# B&R Automation Studio project MotionTestBenchMaster (part 33)

#### HmiVariablesBrowse.st
```iecst
ACTION HmiVariablesBrowse:
	CASE VAR_Level OF
		0:
			memset(ADR(HMI_CFG_Display), 0, SIZEOF(HMI_CFG_Display));
			VAR_Level := 5;

		5:
			VAR_VariableName := VAR_InitialVariableName;

			IF VAR_VariableName <> '' THEN
				VAR_Level := 6;
			ELSE
				IF (AID.DataOut.ProjectType = CST_AID_ProjectMachine) THEN
					HMI_CFG_Display[1].Name := 'CFG_Cap_Par';
					HMI_CFG_Display[1].Visibility := TRUE;
				END_IF

				HMI_CFG_Display[2].Name := 'CFG_ITC';
				HMI_CFG_Display[2].Visibility := TRUE;

				HMI_CFG_Display[10].Name := 'CFG_Par';
				HMI_CFG_Display[10].Visibility := TRUE;
			END_IF

			IF HMI_CFG_Selection <> 0 THEN
				VAR_InitialVariableName := HMI_CFG_Display[HMI_CFG_Selection].Name;
			END_IF

		6:
			VAR_Page := 0;
			VAR_LastElementOld := 0;
			VAR_LastElement := 0;
			VAR_Level := 7;

		7:
			memset(ADR(HMI_CFG_Display), 0, SIZEOF(HMI_CFG_Display));

			IF VAR_InitialVariableName = 'CFG_Par' THEN
				VAR_Level := 8;
			ELSE
				VAR_Level := 9;
			END_IF

		8:
			HMI_CFG_Display[1].Visibility := TRUE;
			HMI_CFG_Display[1].Name := 'CFG_Par';

			VAR_Level := 100;

		9:
			VAR_PV_NinfoState := PV_ninfo(ADR(VAR_VariableName), ADR(VAR_DType), ADR(VAR_Len), ADR(VAR_Dim));

			IF VAR_Dim <= 20 THEN
				FOR var_i := 1 TO VAR_Dim DO
					PV_item(ADR(VAR_VariableName), UDINT_TO_UINT(var_i - 1), ADR(VAR_ItemName));
					strcat(ADR(HMI_CFG_Display[var_i].Name), ADR(VAR_VariableName));
					strcat(ADR(HMI_CFG_Display[var_i].Name), ADR('.'));
					strcat(ADR(HMI_CFG_Display[var_i].Name), ADR(VAR_ItemName));
					HMI_CFG_Display[var_i].Visibility := TRUE;
				END_FOR
			ELSE
				FOR var_i := 1 TO 20 DO
					IF var_i = 1 AND VAR_Page <> 0 THEN
						HMI_CFG_Display[1].Name := 'Previous elements';
						HMI_CFG_Display[1].Visibility := TRUE;
					ELSIF var_i = 20 AND VAR_Dim > INT_TO_UINT(VAR_LastElement) THEN
						HMI_CFG_Display[20].Name := 'Next elements';
						HMI_CFG_Display[20].Visibility := TRUE;
					ELSIF (var_i + (VAR_Page * VAR_LastElementOld)) <= VAR_Dim THEN
						PV_item(ADR(VAR_VariableName), UDINT_TO_UINT((var_i + (VAR_Page * VAR_LastElementOld)) - 1), ADR(VAR_ItemName));
						strcat(ADR(HMI_CFG_Display[var_i].Name), ADR(VAR_VariableName));
						strcat(ADR(HMI_CFG_Display[var_i].Name), ADR('.'));
						strcat(ADR(HMI_CFG_Display[var_i].Name), ADR(VAR_ItemName));
						HMI_CFG_Display[var_i].Visibility := TRUE;
						VAR_LastElement := UDINT_TO_INT(var_i) + (VAR_Page * VAR_LastElementOld);
					END_IF
				END_FOR
			END_IF
			VAR_LastElementOld := VAR_LastElement;

			VAR_Level := 10;

		10:
			IF HMI_CFG_Selection <> 0 AND
				(NOT HMI_CFG_Display[HMI_CFG_Selection].PresentB	AND NOT HMI_CFG_Display[HMI_CFG_Selection].PresentI		AND
				NOT HMI_CFG_Display[HMI_CFG_Selection].PresentR		AND NOT HMI_CFG_Display[HMI_CFG_Selection].PresentSt)	THEN
				IF VAR_Dim <= 20 THEN
					VAR_Level := 15;
				ELSIF HMI_CFG_Selection = 1 AND VAR_Page <> 0 THEN
					VAR_Level := 7;
				ELSIF HMI_CFG_Selection = 20 AND VAR_Dim > INT_TO_UINT(VAR_LastElement) THEN
					VAR_Level := 7;
				ELSE
					VAR_Level := 15;
				END_IF
			END_IF

		15:
			VAR_Page := 0;
			VAR_LastElementOld := 0;
			VAR_LastElement := 0;
			VAR_Level := 16;

		16:
			memset(ADR(HMI_CFG_Display), 0, SIZEOF(HMI_CFG_Display));
			VAR_Level := 20;

		20:
			VAR_PV_NinfoState := PV_ninfo(ADR(VAR_VariableName), ADR(VAR_DType), ADR(VAR_Len), ADR(VAR_Dim));

			IF VAR_DType = 0 THEN
				IF VAR_Dim <= 20 THEN
					FOR var_i := 1 TO VAR_Dim DO
						PV_item(ADR(VAR_VariableName), UDINT_TO_UINT(var_i - 1), ADR(VAR_ItemName));
						strcat(ADR(HMI_CFG_Display[var_i].Name), ADR(VAR_VariableName));
						strcat(ADR(HMI_CFG_Display[var_i].Name), ADR('.'));
						strcat(ADR(HMI_CFG_Display[var_i].Name), ADR(VAR_ItemName));
						HMI_CFG_Display[var_i].Visibility := TRUE;
						VAR_PV_NinfoState := PV_ninfo(ADR(HMI_CFG_Display[var_i].Name), ADR(VAR_DType2), ADR(VAR_Len2), ADR(VAR_Dim2));
						IF VAR_DType2 = 1 THEN
							PV_xgetadr(ADR(HMI_CFG_Display[var_i].Name), ADR(VAR_address), ADR(VAR_Len2));
							memcpy(ADR(HMI_CFG_Display[var_i].ValueB), VAR_address, VAR_Len2);
							HMI_CFG_Display[var_i].PresentB := TRUE;
						ELSIF (VAR_DType2 >= 2 AND VAR_DType2 <= 7) OR VAR_DType2 = 12 THEN
							PV_xgetadr(ADR(HMI_CFG_Display[var_i].Name), ADR(VAR_address), ADR(VAR_Len2));
							memcpy(ADR(HMI_CFG_Display[var_i].ValueI), VAR_address, VAR_Len2);
							HMI_CFG_Display[var_i].PresentI := TRUE;
						ELSIF VAR_DType2 = 8 THEN
							PV_xgetadr(ADR(HMI_CFG_Display[var_i].Name), ADR(VAR_address), ADR(VAR_Len2));
							memcpy(ADR(HMI_CFG_Display[var_i].ValueR), VAR_address, VAR_Len2);
							HMI_CFG_Display[var_i].PresentR := TRUE;
						ELSIF VAR_DType2 = 9 THEN
							PV_xgetadr(ADR(HMI_CFG_Display[var_i].Name), ADR(VAR_address), ADR(VAR_Len2));
							strcpy(ADR(HMI_CFG_Display[var_i].ValueSt), VAR_address);
							HMI_CFG_Display[var_i].PresentSt := TRUE;
						END_IF
					END_FOR
				ELSE
					FOR var_i := 1 TO 20 DO
						IF var_i = 1 AND VAR_Page <> 0 THEN
							HMI_CFG_Display[1].Name := 'Previous elements';
							HMI_CFG_Display[1].Visibility := TRUE;
						ELSIF var_i = 20 AND VAR_Dim > INT_TO_UINT(VAR_LastElement) THEN
							HMI_CFG_Display[20].Name := 'Next elements';
							HMI_CFG_Display[20].Visibility := TRUE;
						ELSIF (var_i + (VAR_Page * VAR_LastElementOld)) <= VAR_Dim THEN
							PV_item(ADR(VAR_VariableName), UDINT_TO_UINT((var_i + (VAR_Page * VAR_LastElementOld)) - 1), ADR(VAR_ItemName));
							strcat(ADR(HMI_CFG_Display[var_i].Name), ADR(VAR_VariableName));
							strcat(ADR(HMI_CFG_Display[var_i].Name), ADR('.'));
							strcat(ADR(HMI_CFG_Display[var_i].Name), ADR(VAR_ItemName));
							HMI_CFG_Display[var_i].Visibility := TRUE;
							VAR_PV_NinfoState := PV_ninfo(ADR(HMI_CFG_Display[var_i].Name), ADR(VAR_DType2), ADR(VAR_Len2), ADR(VAR_Dim2));
							IF VAR_DType2 = 1 THEN
								PV_xgetadr(ADR(HMI_CFG_Display[var_i].Name), ADR(VAR_address), ADR(VAR_Len2));
								memcpy(ADR(HMI_CFG_Display[var_i].ValueB), VAR_address, VAR_Len2);
								HMI_CFG_Display[var_i].PresentB := TRUE;
							ELSIF VAR_DType2 >= 2 AND VAR_DType2 <= 7 OR VAR_DType2 = 12 THEN
								PV_xgetadr(ADR(HMI_CFG_Display[var_i].Name), ADR(VAR_address), ADR(VAR_Len2));
								memcpy(ADR(HMI_CFG_Display[var_i].ValueI), VAR_address, VAR_Len2);
								HMI_CFG_Display[var_i].PresentI := TRUE;
							ELSIF VAR_DType2 = 8 THEN
								PV_xgetadr(ADR(HMI_CFG_Display[var_i].Name), ADR(VAR_address), ADR(VAR_Len2));
								memcpy(ADR(HMI_CFG_Display[var_i].ValueR), VAR_address, VAR_Len2);
								HMI_CFG_Display[var_i].PresentR := TRUE;
							ELSIF VAR_DType2 = 9 THEN
								PV_xgetadr(ADR(HMI_CFG_Display[var_i].Name), ADR(VAR_address), ADR(VAR_Len2));
								strcpy(ADR(HMI_CFG_Display[var_i].ValueSt), VAR_address);
								HMI_CFG_Display[var_i].PresentSt := TRUE;
							END_IF
							VAR_LastElement := UDINT_TO_INT(var_i) + (VAR_Page * VAR_LastElementOld);
						END_IF
					END_FOR
				END_IF
			ELSIF VAR_DType = 15 THEN
				FOR var_i := 1 TO VAR_Dim DO
					strcat(ADR(HMI_CFG_Display[var_i].Name), ADR(VAR_VariableName));
					strcat(ADR(HMI_CFG_Display[var_i].Name), ADR('['));
					itoa((var_i - 1), ADR(VAR_array));
					strcat(ADR(HMI_CFG_Display[var_i].Name), ADR(VAR_array));
					strcat(ADR(HMI_CFG_Display[var_i].Name), ADR(']'));
					HMI_CFG_Display[var_i].Visibility := TRUE;
				END_FOR
			END_IF
			VAR_LastElementOld := VAR_LastElement;

			VAR_Level := 30;

		30:
			IF HMI_CFG_Selection <> 0 AND
				(NOT HMI_CFG_Display[HMI_CFG_Selection].PresentB	AND NOT HMI_CFG_Display[HMI_CFG_Selection].PresentI		AND
				NOT HMI_CFG_Display[HMI_CFG_Selection].PresentR		AND NOT HMI_CFG_Display[HMI_CFG_Selection].PresentSt)	THEN
				IF VAR_Dim <= 20 THEN
					VAR_Level := 15;
				ELSIF HMI_CFG_Selection = 1 AND VAR_Page <> 0 THEN
					VAR_Level := 16;
				ELSIF HMI_CFG_Selection = 20 AND VAR_Dim > INT_TO_UINT(VAR_LastElement) THEN
					VAR_Level := 16;
				ELSE
					VAR_Level := 15;
				END_IF
			END_IF

			FOR var_i := 1 TO 20 DO
				IF HMI_CFG_Display[var_i].PresentB THEN
					PV_xgetadr(ADR(HMI_CFG_Display[var_i].Name), ADR(VAR_address), ADR(VAR_Len2));
					memcpy(VAR_address, ADR(HMI_CFG_Display[var_i].ValueB), VAR_Len2);
				ELSIF HMI_CFG_Display[var_i].PresentI THEN
					PV_xgetadr(ADR(HMI_CFG_Display[var_i].Name), ADR(VAR_address), ADR(VAR_Len2));
					memcpy(VAR_address, ADR(HMI_CFG_Display[var_i].ValueI), VAR_Len2);
				ELSIF HMI_CFG_Display[var_i].PresentR THEN
					PV_xgetadr(ADR(HMI_CFG_Display[var_i].Name), ADR(VAR_address), ADR(VAR_Len2));
					memcpy(VAR_address, ADR(HMI_CFG_Display[var_i].ValueR), VAR_Len2);
				ELSIF HMI_CFG_Display[var_i].PresentSt THEN
					PV_xgetadr(ADR(HMI_CFG_Display[var_i].Name), ADR(VAR_address), ADR(VAR_Len2));
					strcpy(VAR_address, ADR(HMI_CFG_Display[var_i].ValueSt));
				ELSE
					EXIT;
				END_IF
			END_FOR
	END_CASE

	IF EDGENEG(HMI_CFG_Reset) THEN
		IF VAR_Level = 10 OR VAR_Level = 100 THEN
			VAR_InitialVariableName := '';
		END_IF
		VAR_Level := 0;
	END_IF

	IF HMI_CFG_Selection <> 0 THEN
		IF (NOT HMI_CFG_Display[HMI_CFG_Selection].PresentB	AND NOT HMI_CFG_Display[HMI_CFG_Selection].PresentI		AND
			NOT HMI_CFG_Display[HMI_CFG_Selection].PresentR		AND NOT HMI_CFG_Display[HMI_CFG_Selection].PresentSt)	THEN
			IF VAR_Dim <= 20 THEN
				VAR_VariableName := HMI_CFG_Display[HMI_CFG_Selection].Name;
			ELSIF HMI_CFG_Selection = 1 AND VAR_Page <> 0 THEN
				VAR_Page := VAR_Page - 1;
			ELSIF HMI_CFG_Selection = 20 AND VAR_Dim > INT_TO_UINT(VAR_LastElement) THEN
				VAR_Page := VAR_Page + 1;
			ELSE
				VAR_VariableName := HMI_CFG_Display[HMI_CFG_Selection].Name;
			END_IF

			HMI_CFG_Selection := 0;
		END_IF
	END_IF
END_ACTION
```

#### CsvManager.st
```iecst
ACTION CsvManager:
	VAR_FmCmd.FolderCreate		:= FALSE;
	VAR_FmCmd.Load				:= FALSE;
	VAR_FmCmd.Save				:= FALSE;
	VAR_FileName				:= '';

	CFG.DataOut.CapSaved		:= FALSE;
	CFG.DataOut.Busy			:= VAR_CsvMngState <> 800;

	CASE VAR_CsvMngState OF
		0:		//Create Folder
			VAR_FmCmd.FolderCreate := NOT VAR_FmAck.CommandError;

			IF VAR_FmAck.CommandDone THEN
				VAR_CsvMngState := 99;
			END_IF

		99:		//Wait idle
			IF StFmState = 0 AND NOT VAR_FmAck.CommandDone THEN
				VAR_CsvMngState	:= 100;
			END_IF

		100:	//Load machine configuration
			VAR_FmCmd.Load	:= TRUE;
			VAR_FileName	:= 'CFG_PAO.csv';

			FB_MpRecipeCsv.Category	:= ADR(VAR_CategoryConfig);

			IF VAR_FmAck.CommandError THEN
				VAR_CsvMngState			:= 110;
			ELSIF VAR_FmAck.CommandDone AND FB_MpRecipeCsv.Info.LastLoadedRecipe = VAR_FileName THEN
				VAR_CfgPaoName			:= VAR_Header.Name;
				CFG.DataOut.CfgDefault	:= (VAR_Header.Name = 'Default Value');
				VAR_CsvMngState			:= 199;
			END_IF

		110:	//Wait errore reset and idle
			IF NOT VAR_FmAck.CommandError AND StFmState = 0 THEN
				VAR_CsvMngState	:= 115;
			END_IF

		115:	//Save default machine configuration
			VAR_FmCmd.Save			:= TRUE;
			VAR_FileName			:= 'CFG_PAO.csv';
			FB_MpRecipeCsv.Header	:= ADR(CST_DefaultHeader);
			FB_MpRecipeCsv.Category	:= ADR(VAR_CategoryConfig);

			IF VAR_FmAck.CommandError THEN
				CFG.DataOut.ErrorSavingCfg	:= TRUE;
				VAR_CsvMngState				:= 116;
			ELSIF VAR_FmAck.CommandDone THEN
				CFG.DataOut.CfgDefault		:= TRUE;
				VAR_CsvMngState				:= 199;
			END_IF

		116:	//Wait error reset
			IF NOT VAR_FmAck.CommandError THEN
				VAR_CsvMngState	:= 199;
			END_IF

		199:	//Wait idle
			IF StFmState = 0 AND NOT VAR_FmAck.CommandDone THEN
				IF (AID.DataOut.ProjectType = CST_AID_ProjectMachine) THEN
					VAR_CsvMngState	:= 200;
				ELSE
					VAR_CsvMngState	:= 300;
				END_IF
			END_IF

		200:	//Load Hmi configuration
			VAR_FmCmd.Load	:= TRUE;
			VAR_FileName	:= 'HMI_PAO.csv';

			FB_MpRecipeCsv.Category	:= ADR(VAR_CategoryHmi);

			IF VAR_FmAck.CommandError THEN
				VAR_CsvMngState			:= 210;
			ELSIF VAR_FmAck.CommandDone AND FB_MpRecipeCsv.Info.LastLoadedRecipe = VAR_FileName THEN
				VAR_HmiPaoName			:= VAR_Header.Name;
				CFG.DataOut.PaoDefault	:= (VAR_Header.Name = 'Default Value');
				VAR_CsvMngState			:= 299;
			END_IF

		210:	//Wait errore reset and idle
			IF NOT VAR_FmAck.CommandError AND StFmState = 0 THEN
				VAR_CsvMngState	:= 215;
			END_IF

		215:	//Save default Hmi configuration
			VAR_FmCmd.Save			:= TRUE;
			VAR_FileName			:= 'HMI_PAO.csv';
			FB_MpRecipeCsv.Header	:= ADR(CST_DefaultHeader);
			FB_MpRecipeCsv.Category	:= ADR(VAR_CategoryHmi);

			IF VAR_FmAck.CommandError THEN
				CFG.DataOut.ErrorSavingPao	:= TRUE;
				VAR_CsvMngState				:= 216;
			ELSIF VAR_FmAck.CommandDone THEN
				CFG.DataOut.PaoDefault		:= TRUE;
				VAR_CsvMngState				:= 299;
			END_IF

		216:	//Wait error reset
			IF NOT VAR_FmAck.CommandError THEN
				VAR_CsvMngState	:= 299;
			END_IF

		299:	//Wait idle
			IF StFmState = 0 AND NOT VAR_FmAck.CommandDone THEN
				VAR_CsvMngState	:= 300;
			END_IF

		300:	//Load Itc configuration
			VAR_FmCmd.Load	:= TRUE;
			VAR_FileName	:= 'CFG_ITC.csv';

			FB_MpRecipeCsv.Category	:= ADR(VAR_CategoryItc);

			IF VAR_FmAck.CommandError THEN
				VAR_CsvMngState			:= 310;
			ELSIF VAR_FmAck.CommandDone AND FB_MpRecipeCsv.Info.LastLoadedRecipe = VAR_FileName THEN
				VAR_CfgItcName			:= VAR_Header.Name;
				CFG.DataOut.ItcDefault	:= (VAR_Header.Name = 'Default Value');
				VAR_CsvMngState			:= 399;
			END_IF

		310:	//Wait errore reset and idle
			IF NOT VAR_FmAck.CommandError AND StFmState = 0 THEN
				VAR_CsvMngState	:= 315;
			END_IF

		315:	//Save default Itc configuration
			VAR_FmCmd.Save			:= TRUE;
			VAR_FileName			:= 'CFG_ITC.csv';
			FB_MpRecipeCsv.Header	:= ADR(CST_DefaultHeader);
			FB_MpRecipeCsv.Category	:= ADR(VAR_CategoryItc);

			IF VAR_FmAck.CommandError THEN
				CFG.DataOut.ErrorSavingItc	:= TRUE;
				VAR_CsvMngState				:= 316;
			ELSIF VAR_FmAck.CommandDone THEN
				CFG.DataOut.ItcDefault		:= TRUE;
				VAR_CsvMngState				:= 399;
			END_IF

		316:	//Wait error reset
			IF NOT VAR_FmAck.CommandError THEN
				VAR_CsvMngState	:= 399;
			END_IF

		399:	//Wait idle
			IF StFmState = 0 AND NOT VAR_FmAck.CommandDone THEN
				IF (AID.DataOut.ProjectType = CST_AID_ProjectMachine) THEN
					IF CFG_Par.Machine.Type.SRMA THEN
						VAR_CsvMngState	:= 500;
					ELSIF CFG_Par.Machine.Type.SRMB OR CFG_Par.Machine.Type.SRMC OR CFG_Par.Machine.Type.SRMH OR CFG_Par.Machine.Type.SRMO THEN
						VAR_CsvMngState	:= 400;
					ELSIF CFG_Par.Machine.Type.SRME THEN
						VAR_CsvMngState	:= 500;
					END_IF
				ELSE
					VAR_CsvMngState	:= 700;
				END_IF
			END_IF

		400:	//Load Cap configuration
			VAR_FmCmd.Load	:= TRUE;
			VAR_FileName	:= 'CFG_CAP.csv';

			FB_MpRecipeCsv.Category	:= ADR(VAR_CategoryCfgCap);

			IF VAR_FmAck.CommandError THEN
				VAR_CsvMngState				:= 410;
			ELSIF VAR_FmAck.CommandDone AND FB_MpRecipeCsv.Info.LastLoadedRecipe = VAR_FileName THEN
				VAR_CfgCapName				:= VAR_Header.Name;
				CFG.DataOut.CfgCapDefault	:= (VAR_Header.Name = 'Default Value');
				VAR_CsvMngState				:= 499;
			END_IF

		410:	//Wait errore reset and idle
			IF NOT VAR_FmAck.CommandError AND StFmState = 0 THEN
				VAR_CsvMngState	:= 415;
			END_IF

		415:	//Save default Cap configuration
			VAR_FmCmd.Save			:= TRUE;
			VAR_FileName			:= 'CFG_CAP.csv';
			FB_MpRecipeCsv.Header	:= ADR(CST_DefaultHeader);
			FB_MpRecipeCsv.Category	:= ADR(VAR_CategoryCfgCap);

			IF VAR_FmAck.CommandError THEN
				CFG.DataOut.ErrorSavingCfgCap	:= TRUE;
				VAR_CsvMngState					:= 416;
			ELSIF VAR_FmAck.CommandDone THEN
				CFG.DataOut.CfgCapDefault		:= TRUE;
				VAR_CsvMngState					:= 499;
			END_IF

		416:	//Wait error reset
			IF NOT VAR_FmAck.CommandError THEN
				VAR_CsvMngState	:= 499;
			END_IF

		499:	//Wait idle
			IF StFmState = 0 AND NOT VAR_FmAck.CommandDone THEN
				VAR_CsvMngState	:= 500;
			END_IF

		500:	//Load Motion configuration
			VAR_FmCmd.Load	:= TRUE;
			VAR_FileName	:= 'CFG_MC.csv';

			FB_MpRecipeCsv.Category	:= ADR(VAR_CategoryMotion);

			IF VAR_FmAck.CommandError THEN
				VAR_CsvMngState			:= 510;
			ELSIF VAR_FmAck.CommandDone AND FB_MpRecipeCsv.Info.LastLoadedRecipe = VAR_FileName THEN
				VAR_CfgMotionName			:= VAR_Header.Name;
				CFG.DataOut.MotionDefault	:= (VAR_Header.Name = 'Default Value');
				VAR_CsvMngState				:= 599;
			END_IF

		510:	//Wait errore reset and idle
			IF NOT VAR_FmAck.CommandError AND StFmState = 0 THEN
				VAR_CsvMngState	:= 515;
			END_IF

		515:	//Save default Motion configuration
			VAR_FmCmd.Save			:= TRUE;
			VAR_FileName			:= 'CFG_MC.csv';
			FB_MpRecipeCsv.Header	:= ADR(CST_DefaultHeader);
			FB_MpRecipeCsv.Category	:= ADR(VAR_CategoryMotion);

			IF VAR_FmAck.CommandError THEN
				CFG.DataOut.ErrorSavingMotion	:= TRUE;
				VAR_CsvMngState					:= 516;
			ELSIF VAR_FmAck.CommandDone THEN
				CFG.DataOut.MotionDefault	:= TRUE;
				VAR_CsvMngState				:= 599;
			END_IF

		516:	//Wait error reset
			IF NOT VAR_FmAck.CommandError THEN
				VAR_CsvMngState	:= 599;
			END_IF

		599:	//Wait idle
			IF StFmState = 0 AND NOT VAR_FmAck.CommandDone THEN
				IF CFG_Par.Machine.Type.SRMA THEN
					VAR_CsvMngState	:= 600;
				ELSIF CFG_Par.Machine.Type.SRMB OR CFG_Par.Machine.Type.SRMC OR CFG_Par.Machine.Type.SRMH OR CFG_Par.Machine.Type.SRMO THEN
					VAR_CsvMngState	:= 600;
				ELSIF CFG_Par.Machine.Type.SRME THEN
					VAR_CsvMngState	:= 700;
				END_IF
			END_IF

		600:	//Load Ops configuration
			VAR_FmCmd.Load	:= TRUE;
			VAR_FileName	:= 'CFG_OPS.csv';

			FB_MpRecipeCsv.Category	:= ADR(VAR_CategoryCfgDoor);

			IF VAR_FmAck.CommandError THEN
				VAR_CsvMngState			:= 610;
			ELSIF VAR_FmAck.CommandDone AND FB_MpRecipeCsv.Info.LastLoadedRecipe = VAR_FileName THEN
				VAR_CfgDoorName			:= VAR_Header.Name;
				CFG.DataOut.OPSDefault	:= (VAR_Header.Name = 'Default Value');
				VAR_CsvMngState				:= 699;
			END_IF

		610:	//Wait errore reset and idle
			IF NOT VAR_FmAck.CommandError AND StFmState = 0 THEN
				VAR_CsvMngState	:= 615;
			END_IF

		615:	//Save default OPS configuration
			VAR_FmCmd.Save			:= TRUE;
			VAR_FileName			:= 'CFG_OPS.csv';
			FB_MpRecipeCsv.Header	:= ADR(CST_DefaultHeader);
			FB_MpRecipeCsv.Category	:= ADR(VAR_CategoryCfgDoor);

			IF VAR_FmAck.CommandError THEN
				CFG.DataOut.ErrorSavingOPS	:= TRUE;
				VAR_CsvMngState					:= 616;
			ELSIF VAR_FmAck.CommandDone THEN
				CFG.DataOut.OPSDefault	:= TRUE;
				VAR_CsvMngState				:= 699;
			END_IF

		616:	//Wait error reset
			IF NOT VAR_FmAck.CommandError THEN
				VAR_CsvMngState	:= 699;
			END_IF

		699:	//Wait idle
			IF StFmState = 0 AND NOT VAR_FmAck.CommandDone THEN
				VAR_CsvMngState	:= 700;
			END_IF

		700:	//Check for error
			IF CFG.DataOut.ErrorSavingCfg OR CFG.DataOut.ErrorSavingItc OR ((CFG.DataOut.ErrorSavingPao OR CFG.DataOut.ErrorSavingCfgCap OR CFG.DataOut.ErrorSavingMotion OR CFG.DataOut.OPSDefault) AND AID.DataOut.ProjectType = CST_AID_ProjectMachine) THEN
				VAR_CsvMngState		:= 9998;
			ELSIF CFG.DataOut.CfgDefault OR CFG.DataOut.ItcDefault OR ((CFG.DataOut.PaoDefault OR CFG.DataOut.CfgCapDefault OR CFG.DataOut.MotionDefault OR CFG.DataOut.OPSDefault) AND AID.DataOut.ProjectType = CST_AID_ProjectMachine) THEN
				VAR_CsvMngState		:= 9999;
			ELSE
				IF (VAR_CfgPaoName = VAR_CfgItcName) AND (((VAR_CfgPaoName = VAR_HmiPaoName) AND (VAR_CfgPaoName = VAR_CfgMotionName) AND
					((VAR_CfgPaoName = VAR_CfgDoorName) OR CFG_Par.Machine.Type.SRME)) OR AID.DataOut.ProjectType = CST_AID_ProjectSkid) THEN
					HMI_MachineId	:= VAR_CfgPaoName;
				ELSE
					HMI_MachineId	:= 'Error Name';
				END_IF
				VAR_CsvMngState		:= 800;
			END_IF

		800:	//Initial Configuration done - Waiting for request
			CFG.DataOut.ConfigLoaded := TRUE;

			IF HMI_PB[PB_CFG_LoadPao].ON THEN
				VAR_CsvMngState		:= 1000;
			ELSIF HMI_PB[PB_CFG_SavePao].ON THEN
				VAR_CsvMngState		:= 1050;
			ELSIF HMI_PB[PB_CFG_LoadCfg].ON THEN
				IF VAR_InitialVariableName = 'CFG_ITC' THEN
					VAR_CsvMngState	:= 1100;
				ELSIF VAR_InitialVariableName = 'CFG_Cap_Par' THEN
					VAR_CsvMngState	:= 1200;
				ELSIF VAR_InitialVariableName = 'CFG_Par' THEN
					VAR_CsvMngState	:= 1300;
				END_IF
			ELSIF HMI_PB[PB_CFG_SaveCfg].ON THEN
				IF VAR_InitialVariableName = 'CFG_ITC' THEN
					VAR_CsvMngState	:= 1150;
				ELSIF VAR_InitialVariableName = 'CFG_Cap_Par' THEN
					VAR_CsvMngState	:= 1250;
				ELSIF VAR_InitialVariableName = 'CFG_Par' THEN
					VAR_CsvMngState	:= 1350;
				END_IF
			ELSIF CAP.DataOut.ConfigSaveReq THEN
				VAR_CsvMngState	:= 1250;
			ELSIF OPS.DataOut.ConfigSaveReq THEN
				VAR_CsvMngState	:= 1450;
			END_IF

		1000:	//Manual - Load Hmi configuration
			VAR_FmCmd.Load	:= TRUE;
			VAR_FileName	:= 'HMI_PAO.csv';

			FB_MpRecipeCsv.Category	:= ADR(VAR_CategoryHmi);

			IF VAR_FmAck.CommandError OR VAR_FmAck.CommandDone THEN
				VAR_CsvMngState := 1010;
			END_IF

		1010:	//Wait errore reset and idle
			IF NOT VAR_FmAck.CommandError AND StFmState = 0 AND NOT HMI_PB[PB_CFG_LoadPao].ON THEN
				VAR_CsvMngState	:= 800;
			END_IF

		1050:	//Manual - Save Hmi configuration
			VAR_FmCmd.Save			:= TRUE;
			VAR_FileName			:= 'HMI_PAO.csv';
			VAR_Header.Name			:= HMI_MachineId;
			FB_MpRecipeCsv.Category	:= ADR(VAR_CategoryHmi);

			IF VAR_FmAck.CommandError OR VAR_FmAck.CommandDone THEN
				VAR_CsvMngState	:= 1060;
			END_IF

		1060:	//Wait errore reset and idle
			IF NOT VAR_FmAck.CommandError AND StFmState = 0 AND NOT HMI_PB[PB_CFG_SavePao].ON THEN
				VAR_CsvMngState	:= 800;
			END_IF

		1100:	//Manual - Load ITC configuration
			VAR_FmCmd.Load	:= TRUE;
			VAR_FileName	:= 'CFG_ITC.csv';

			FB_MpRecipeCsv.Category	:= ADR(VAR_CategoryItc);

			IF VAR_FmAck.CommandError OR VAR_FmAck.CommandDone THEN
				VAR_CsvMngState := 1110;
			END_IF

		1110:	//Wait errore reset and idle
			IF NOT VAR_FmAck.CommandError AND StFmState = 0 AND NOT HMI_PB[PB_CFG_LoadCfg].ON THEN
				VAR_CsvMngState	:= 800;
			END_IF

		1150:	//Manual - Save ITC configuration
			VAR_FmCmd.Save			:= TRUE;
			VAR_FileName			:= 'CFG_ITC.csv';
			VAR_Header.Name			:= HMI_MachineId;
			FB_MpRecipeCsv.Category	:= ADR(VAR_CategoryItc);

			IF VAR_FmAck.CommandError OR VAR_FmAck.CommandDone THEN
				VAR_CsvMngState	:= 1160;
			END_IF

		1160:	//Wait errore reset and idle
			IF NOT VAR_FmAck.CommandError AND StFmState = 0 AND NOT HMI_PB[PB_CFG_SaveCfg].ON THEN
				VAR_CsvMngState	:= 800;
			END_IF

		1200:	//Manual - Load Hmi configuration
			VAR_FmCmd.Load	:= TRUE;
			VAR_FileName	:= 'CFG_CAP.csv';

			FB_MpRecipeCsv.Category	:= ADR(VAR_CategoryCfgCap);

			IF VAR_FmAck.CommandError OR VAR_FmAck.CommandDone THEN
				VAR_CsvMngState := 1210;
			END_IF

		1210:	//Wait errore reset and idle
			IF NOT VAR_FmAck.CommandError AND StFmState = 0 AND NOT HMI_PB[PB_CFG_LoadCfg].ON THEN
				VAR_CsvMngState	:= 800;
			END_IF

		1250:	//Manual - Save Hmi configuration
			VAR_FmCmd.Save			:= TRUE;
			VAR_FileName			:= 'CFG_CAP.csv';
			VAR_Header.Name			:= HMI_MachineId;
			FB_MpRecipeCsv.Category	:= ADR(VAR_CategoryCfgCap);

			IF VAR_FmAck.CommandError OR VAR_FmAck.CommandDone THEN
				VAR_CsvMngState	:= 1260;
			END_IF

		1260:	//Wait errore reset and idle
			CFG.DataOut.CapSaved	:= TRUE;

			IF NOT VAR_FmAck.CommandError AND StFmState = 0 AND NOT HMI_PB[PB_CFG_SaveCfg].ON AND NOT CAP.DataOut.ConfigSaveReq THEN
				VAR_CsvMngState	:= 800;
			END_IF

		1300:	//Manual - Load Hmi configuration
			VAR_FmCmd.Load	:= TRUE;
			VAR_FileName	:= 'CFG_PAO.csv';

			FB_MpRecipeCsv.Category	:= ADR(VAR_CategoryConfig);

			IF VAR_FmAck.CommandError OR VAR_FmAck.CommandDone THEN
				VAR_CsvMngState := 1310;
			END_IF

		1310:	//Wait errore reset and idle
			IF NOT VAR_FmAck.CommandError AND StFmState = 0 AND NOT HMI_PB[PB_CFG_LoadCfg].ON THEN
				VAR_CsvMngState	:= 800;
			END_IF

		1350:	//Manual - Save Hmi configuration
			VAR_FmCmd.Save			:= TRUE;
			VAR_FileName			:= 'CFG_PAO.csv';
			VAR_Header.Name			:= HMI_MachineId;
			FB_MpRecipeCsv.Category	:= ADR(VAR_CategoryConfig);

			IF VAR_FmAck.CommandError OR VAR_FmAck.CommandDone THEN
				VAR_CsvMngState	:= 1360;
			END_IF

		1360:	//Wait errore reset and idle
			IF NOT VAR_FmAck.CommandError AND StFmState = 0 AND NOT HMI_PB[PB_CFG_SaveCfg].ON THEN
				VAR_CsvMngState	:= 800;
			END_IF

		1450:	//Manual - Save Hmi configuration
			VAR_FmCmd.Save			:= TRUE;
			VAR_FileName			:= 'CFG_OPS.csv';
			VAR_Header.Name			:= HMI_MachineId;
			FB_MpRecipeCsv.Category	:= ADR(VAR_CategoryCfgDoor);

			IF VAR_FmAck.CommandError OR VAR_FmAck.CommandDone THEN
				VAR_CsvMngState	:= 1460;
			END_IF

		1460:	//Wait errore reset and idle
			CFG.DataOut.OpsSaved	:= TRUE;

			IF NOT VAR_FmAck.CommandError AND StFmState = 0 AND NOT CAP.DataOut.ConfigSaveReq THEN
				VAR_CsvMngState	:= 800;
			END_IF

		9998:	// Error saving file

		9999:	// Default configuration loaded
	END_CASE
END_ACTION
```

#### FileManager.st
```iecst
ACTION FileManager:
	CASE StFmState OF
		0:		//Wait command
			FB_MpRecipeCsv.LoadType		:= mpRECIPE_CSV_LOAD_ALL;
			FB_MpRecipeCsv.Load			:= FALSE;
			FB_MpRecipeCsv.Save			:= FALSE;
			FB_MpRecipeCsv.ErrorReset	:= FALSE;

			VAR_FmAck.CommandBusy	:= FALSE;
			VAR_FmAck.CommandDone	:= FALSE;
			VAR_FmAck.CommandError	:= FALSE;

			IF FB_MpRecipeCsv.Error THEN
				StFmState	:= 999;
			ELSIF VAR_FmCmd.FolderCreate THEN
				StFmState	:= 100;
			ELSIF VAR_FmCmd.Load THEN
				StFmState	:= 200;
			ELSIF VAR_FmCmd.Save THEN
				StFmState	:= 250;
			END_IF

		100:	//Create Folder
			VAR_FmAck.CommandBusy	:= NOT(VAR_FmAck.CommandDone OR VAR_FmAck.CommandError);

			IF NOT VAR_FmCmd.FolderCreate THEN
				StFmState	:= 0;
			ELSIF VAR_FmAck.CommandBusy THEN
				FB_DirCreate();

				IF FB_DirCreate.status = ERR_OK OR FB_DirCreate.status = fiERR_DIR_ALREADY_EXIST THEN
					VAR_FmAck.CommandDone	:= TRUE;
				ELSIF FB_DirCreate.status <> ERR_FUB_BUSY AND FB_DirCreate.status <> ERR_FUB_ENABLE_FALSE THEN
					VAR_FmAck.CommandError	:= TRUE;
					VAR_FmAck.ErrorCode		:= FB_DirCreate.status;
					VAR_FmAck.ErroreState	:= ERR_FOLDER_CREATE;
				END_IF
			END_IF

		200:	//Load
			VAR_FmAck.CommandBusy	:= NOT(VAR_FmAck.CommandDone OR VAR_FmAck.CommandError);
			FB_MpRecipeCsv.Load		:= TRUE;

			IF EDGEPOS(FB_MpRecipeCsv.Error) THEN
				VAR_FmAck.CommandError	:= TRUE;
				VAR_FmAck.ErrorCode		:= FB_MpRecipeCsv.Info.Diag.StatusID.Code;
				VAR_FmAck.ErroreState	:= ERR_LOAD;
			ELSIF EDGEPOS(FB_MpRecipeCsv.CommandDone) AND NOT FB_MpRecipeCsv.Error THEN
				VAR_FmAck.CommandDone	:= TRUE;
			ELSIF NOT VAR_FmCmd.Load AND (NOT FB_MpRecipeCsv.CommandBusy OR FB_MpRecipeCsv.Error) THEN
				StFmState	:= 0;
			END_IF

		250:	//Save configuration
			VAR_FmAck.CommandBusy	:= NOT(VAR_FmAck.CommandDone OR VAR_FmAck.CommandError);
			FB_MpRecipeCsv.Save		:= TRUE;

				IF EDGEPOS(FB_MpRecipeCsv.Error) THEN
					VAR_FmAck.CommandError	:= TRUE;
					VAR_FmAck.ErrorCode		:= FB_MpRecipeCsv.Info.Diag.StatusID.Code;
					VAR_FmAck.ErroreState	:= ERR_SAVE;
				ELSIF EDGEPOS(FB_MpRecipeCsv.CommandDone) AND NOT FB_MpRecipeCsv.Error THEN
					VAR_FmAck.CommandDone	:= TRUE;
				ELSIF NOT VAR_FmCmd.Save AND (NOT FB_MpRecipeCsv.CommandBusy OR FB_MpRecipeCsv.Error) THEN
					StFmState	:= 0;
				END_IF

		999:	//Error Reset
			FB_MpRecipeCsv.ErrorReset := TRUE;

			IF NOT FB_MpRecipeCsv.Error THEN
				StFmState	:= 0;
			END_IF

	END_CASE
END_ACTION
```

### Package Logical/30_MC - Motion Main Folder

### GlobalVariables.var
```iecst
(*General axis task global interface*)
VAR
	VAR_Machine : ST_Machine;
END_VAR
(*Simulation Variables*)
VAR
	VAR_SimulationOn : BOOL;
END_VAR
(*Machine Master Fast*)
VAR
	fbMachineMasterFast : FB_MasterAxis;
END_VAR
(*Master Module Axis Declaration*)
VAR
	VAR_AxPowerSupply01 : ACP10AXIS_typ;
	VAR_AxPowerSupply02 : ACP10AXIS_typ;
	VAR_AxMachineMaster : ACP10AXIS_typ;
END_VAR
(*Filler Module Axis Declaration*)
VAR
	VAR_AxEncEmul : ACP10AXIS_typ;
	VAR_AxFillerModuleMaster : ACP10AXIS_typ;
	VAR_AxFillerIn10 : ACP10AXIS_typ;
	VAR_AxFillerIn09 : ACP10AXIS_typ;
	VAR_AxFillerIn08 : ACP10AXIS_typ;
	VAR_AxFillerIn07 : ACP10AXIS_typ;
	VAR_AxFillerIn06 : ACP10AXIS_typ;
	VAR_AxFillerIn05 : ACP10AXIS_typ;
	VAR_AxFillerIn04 : ACP10AXIS_typ;
	VAR_AxFillerIn03 : ACP10AXIS_typ;
	VAR_AxFillerIn02 : ACP10AXIS_typ;
	VAR_AxFillerIn01 : ACP10AXIS_typ;
	VAR_AxFillerMain : ACP10AXIS_typ;
	VAR_AxFillerOut01 : ACP10AXIS_typ;
	VAR_AxFillerOut02 : ACP10AXIS_typ;
	VAR_AxFillerOut03 : ACP10AXIS_typ;
	VAR_AxFillerOut04 : ACP10AXIS_typ;
	VAR_AxFillerOut05 : ACP10AXIS_typ;
	VAR_AxFillerOut06 : ACP10AXIS_typ;
END_VAR
(*Inlet Module Axis Declaration*)
VAR
	VAR_AxInletModuleMaster : ACP10AXIS_typ;
	VAR_AxInletIn04 : ACP10AXIS_typ;
	VAR_AxInletIn03 : ACP10AXIS_typ;
	VAR_AxInletIn02 : ACP10AXIS_typ;
	VAR_AxInletIn01 : ACP10AXIS_typ;
	VAR_AxInletMain : ACP10AXIS_typ;
	VAR_AxInletOut01 : ACP10AXIS_typ;
	VAR_AxInletOut02 : ACP10AXIS_typ;
	VAR_AxInletOut03 : ACP10AXIS_typ;
	VAR_AxInletOut04 : ACP10AXIS_typ;
END_VAR
(*Outlet Module Axis Declaration*)
VAR
	VAR_AxOutletModuleMaster : ACP10AXIS_typ;
	VAR_AxOutletIn04 : ACP10AXIS_typ;
	VAR_AxOutletIn03 : ACP10AXIS_typ;
	VAR_AxOutletIn02 : ACP10AXIS_typ;
	VAR_AxOutletIn01 : ACP10AXIS_typ;
	VAR_AxOutletMain : ACP10AXIS_typ;
	VAR_AxOutletOut01 : ACP10AXIS_typ;
	VAR_AxOutletOut02 : ACP10AXIS_typ;
	VAR_AxOutletOut03 : ACP10AXIS_typ;
	VAR_AxOutletOut04 : ACP10AXIS_typ;
END_VAR
(*Modules mapp link*)
VAR
	VAR_SpareLink : MpComIdentType; (*Mapp link to spare axes*)
	VAR_MachineLink : MpComIdentType; (*Mapp link for machine*)
	VAR_MasterModuleLink : MpComIdentType; (*Mapp link for master module*)
	VAR_FillerModuleLink : MpComIdentType; (*Mapp link for filler module*)
	VAR_InletModuleLink : MpComIdentType; (*Mapp link for outlet module*)
	VAR_OutletModuleLink : MpComIdentType; (*Mapp link for outlet module*)
	VAR_MpComLinkToParentSpare : UDINT;
END_VAR
(*DECELERATION*)
VAR
	VAR_EmergencyDec : REAL;
	VAR_ShutDownDec : REAL;
END_VAR
(*CAM*)
VAR
	VAR_xMachineInitDone : BOOL;
	VAR_xInletInitDone : BOOL;
	VAR_xFillerInitDone : BOOL;
	VAR_xOutletInitDone : BOOL;
	VAR_CamInitialized : BOOL; (*//v4.A.A.1.6.7*)
END_VAR
(*INTERCHANGE MOTION*)
VAR
	ITC_Motion : ST_LabellerMotionInterface;
END_VAR
```

### CamConfigurator.var
```iecst
(*Cam Configurator*)
(*Clock A-B*)
VAR CONSTANT
	CST_SubModuleMachineCk : USINT := CST_MasterSubModule; (*0 - Master; 1 - Filler; 2 - Outlet*)
	CST_AxisMachineCk : USINT := CST_ModuleMasterAxis;
	CST_OnPositionCkA : REAL := 0.0;
	CST_OffPositionCkA : REAL := 180.0;
	CST_OnPositionCkB : REAL := 270.0;
	CST_OffPositionCkB : REAL := 90.0;
	CST_OnPositionCkA_Fma : REAL := 10.0;
	CST_OffPositionCkA_Fma : REAL := 190.0;
	CST_OnPositionCkB_Fma : REAL := 100.0;
	CST_OffPositionCkB_Fma : REAL := 280.0;
	CST_AdvTimeCkA : REAL := 0.0;
END_VAR
(*Clock 02*)
VAR CONSTANT
	CST_SubModuleCk02 : USINT := CST_MasterSubModule; (*0 - Master; 1 - Filler; 2 - Outlet*)
	CST_AxisCk02 : USINT := CST_ModuleMasterAxis;
	CST_OnPositionCk02 : REAL := 10.0;
	CST_OffPositionCk02 : REAL := 15.0;
	CST_AdvTimeCk02 : REAL := 0.0;
END_VAR
(*Clock 03*)
VAR CONSTANT
	CST_SubModuleCk03 : USINT := CST_MasterSubModule; (*0 - Master; 1 - Filler; 2 - Outlet*)
	CST_AxisCk03 : USINT := CST_ModuleMasterAxis;
	CST_OnPositionCk03 : REAL := 10.0;
	CST_OffPositionCk03 : REAL := 20.0;
	CST_AdvTimeCk03 : REAL := 0.0;
END_VAR
(*Clock 04*)
VAR CONSTANT
	CST_SubModuleCk04 : USINT := CST_MasterSubModule; (*0 - Master; 1 - Filler; 2 - Outlet*)
	CST_AxisCk04 : USINT := CST_ModuleMasterAxis;
	CST_OnPositionCk04 : REAL := 20.0;
	CST_OffPositionCk04 : REAL := 30.0;
	CST_AdvTimeCk04 : USINT := 0;
END_VAR
(*Clock 05*)
VAR CONSTANT
	CST_SubModuleCk05 : USINT := CST_MasterSubModule; (*0 - Master; 1 - Filler; 2 - Outlet*)
	CST_AxisCk05 : USINT := CST_ModuleMasterAxis;
	CST_OnPositionCk05 : REAL := 20.0;
	CST_OffPositionCk05 : REAL := 40.0;
	CST_AdvTimeCk05 : REAL := 0.0;
END_VAR
(*Clock 06*)
VAR CONSTANT
	CST_SubModuleCk06 : USINT := CST_MasterSubModule; (*0 - Master; 1 - Filler; 2 - Outlet*)
	CST_AxisCk06 : USINT := CST_ModuleMasterAxis;
	CST_OnPositionCk06 : REAL := 30.0;
	CST_OffPositionCk06 : REAL := 60.0;
	CST_AdvTimeCk06 : REAL := 0.0;
END_VAR
(*Clock 07*)
VAR CONSTANT
	CST_SubModuleCk07 : USINT := CST_MasterSubModule; (*0 - Master; 1 - Filler; 2 - Outlet*)
	CST_AxisCk07 : USINT := CST_ModuleMasterAxis;
	CST_OnPositionCk07 : REAL := 60.0;
	CST_OffPositionCk07 : REAL := 30.0;
	CST_AdvTimeCk07 : REAL := 0.0;
END_VAR
(*Clock 08*)
VAR CONSTANT
	CST_SubModuleCk08 : USINT := CST_MasterSubModule; (*0 - Master; 1 - Filler; 2 - Outlet*)
	CST_AxisCk08 : USINT := CST_ModuleMasterAxis;
	CST_OnPositionCk08 : REAL := 60.0;
	CST_OffPositionCk08 : REAL := 30.0;
	CST_AdvTimeCk08 : REAL := 0.0;
END_VAR
```

### MotionPermanent.var
```iecst
(*Master Module*)
VAR RETAIN
	VAR_PowerSupplyHomeData : ST_AxisHome;
	VAR_AxMachineMasterHomeData : ST_AxisHome;
	VAR_AbsEncPerm : ST_AbsEncPerm;
END_VAR
(*Filler Module*)
VAR RETAIN
	VAR_FillerMasterHomeData : ST_AxisHome;
	VAR_FillerMainHomeData : ST_AxisHome;
	VAR_FillerIn01HomeData : ST_AxisHome;
	VAR_FillerIn02HomeData : ST_AxisHome;
	VAR_FillerIn03HomeData : ST_AxisHome;
	VAR_FillerIn04HomeData : ST_AxisHome;
	VAR_FillerIn05HomeData : ST_AxisHome;
	VAR_FillerIn06HomeData : ST_AxisHome;
	VAR_FillerIn07HomeData : ST_AxisHome;
	VAR_FillerIn08HomeData : ST_AxisHome;
	VAR_FillerIn09HomeData : ST_AxisHome;
	VAR_FillerIn10HomeData : ST_AxisHome;
	VAR_FillerOut01HomeData : ST_AxisHome;
	VAR_FillerOut02HomeData : ST_AxisHome;
	VAR_FillerOut03HomeData : ST_AxisHome;
	VAR_FillerOut04HomeData : ST_AxisHome;
	VAR_FillerOut05HomeData : ST_AxisHome;
	VAR_FillerOut06HomeData : ST_AxisHome;
END_VAR
(*Outlet Module*)
VAR RETAIN
	VAR_OutletMasterHomeData : ST_AxisHome;
	VAR_OutletIn01HomeData : ST_AxisHome;
	VAR_OutletIn02HomeData : ST_AxisHome;
	VAR_OutletIn03HomeData : ST_AxisHome;
	VAR_OutletIn04HomeData : ST_AxisHome;
	VAR_OutletMainHomeData : ST_AxisHome;
	VAR_OutletOut01HomeData : ST_AxisHome;
	VAR_OutletOut02HomeData : ST_AxisHome;
	VAR_OutletOut03HomeData : ST_AxisHome;
	VAR_OutletOut04HomeData : ST_AxisHome;
END_VAR
(*Inlet Module*)
VAR RETAIN
	VAR_InletMasterHomeData : ST_AxisHome;
	VAR_InletIn01HomeData : ST_AxisHome;
	VAR_InletIn02HomeData : ST_AxisHome;
	VAR_InletIn03HomeData : ST_AxisHome;
	VAR_InletIn04HomeData : ST_AxisHome;
	VAR_InletMainHomeData : ST_AxisHome;
	VAR_InletOut01HomeData : ST_AxisHome;
	VAR_InletOut02HomeData : ST_AxisHome;
	VAR_InletOut03HomeData : ST_AxisHome;
	VAR_InletOut04HomeData : ST_AxisHome;
END_VAR
```

### ToConfigureConstant.var
```iecst
(*Absolute Position Constant*)
VAR CONSTANT
	CST_StepsAbsolutePositionFiller : UINT := 10; (*Number Of Steps Carousel Unit*)
	CST_StepsAbsolutePositionOutlet : UINT := 10; (*Number Of Steps*)
	CST_StepsAbsolutePositionInlet : UINT := 10; (*Number Of Steps*)
	CST_AxesMultiplexingOn : BOOL := TRUE; (*V4.A.A.1.6.10 (replace CFG_MC.Generic.AxesMultiplexingOn with CST_AxesMultiplexingOn)*)
END_VAR
```

### Package Logical/30_MC/AxisTable - Package

### Data object Logical/30_MC/AxisTable/acp10etxen (Ett)

- acp10etxen.ett (not shown)

### Package Logical/30_MC/AxisTable/VirtualTables - Package

### Data object Logical/30_MC/AxisTable/VirtualTables/gVirtualPr (Apt) - ACOPOS Parameter Table

#### gVirtPar.apt
```
AcoposParameterTable:
  Root Parameters:
    351 = 0 (Name=ERRESP_UDC_POWERFAIL)  // Power mains: Error response
    80 = 1 (Name=PHASE_MON_IGNORE, Disabled=TRUE)  // Power mains: Ignore phase failure
    368 = 0 (Name=UVLIM_MODE)  // CTRL DC bus: Limiter: Mode
    COMBI SYNCHRONIZATION:
      777 = VAR_I4_0+0 (Name=FUNCTION_BLOCK_CREATE)  // Function block: Create a FB instance
      777 = IPL_MODE+0 (Name=FUNCTION_BLOCK_CREATE)  // Function block: Create a FB instance
      777 = CURVE_MODE+0 (Name=FUNCTION_BLOCK_CREATE)  // Function block: Create a FB instance
      777 = CURVE_MODE+1 (Name=FUNCTION_BLOCK_CREATE)  // Function block: Create a FB instance
      777 = CURVE_MODE+3 (Name=FUNCTION_BLOCK_CREATE)  // Function block: Create a FB instance
      777 = CURVE_MODE+4 (Name=FUNCTION_BLOCK_CREATE)  // Function block: Create a FB instance
      777 = CURVE_MODE+5 (Name=FUNCTION_BLOCK_CREATE)  // Function block: Create a FB instance
      777 = ARITH_MODE+0 (Name=FUNCTION_BLOCK_CREATE)  // Function block: Create a FB instance
      VAR:
        4096 = 0 (Name=VAR_I4_0+0)  // FB0 VAR I4 variable0
        4120 = 0 (Name=VAR_I4_3+0)  // FB0 FB VAR: Variable3 I4
      IPL:
        8704 = 0 (Name=IPL_MODE+0)  // FB0 IPL Mode
        8712 = VAR_I4_0+0 (Name=IPL_IN_PARID+0)  // FB0 IPL Parameter ID of input
        8760 = 0 (Name=IPL_EV_PARID+0)  // FB0 IPL Parameter ID of event input
        8720 = 800 (Name=IPL_CYCLE_TIME+0, Unit=us)  // FB0 IPL Cycle time
        8728 = 400 (Name=IPL_EXTRAPOLATION_TIME+0, Unit=us)  // FB0 IPL Extrapolation time
        8704 = 1 (Name=IPL_MODE+0)  // FB0 IPL Mode = LINEAR INTERPOLATION
      CURVE 0:
        8192 = 0 (Name=CURVE_MODE+0)  // FB0 CURVE Mode
        8200 = IPL_VALUE_I4+0 (Name=CURVE_IN_PARID+0)  // FB0 CURVE Parameter ID of input
        8208 = 65535 (Name=CURVE_AUT_DATA_INDEX+0)  // FB0 CURVE Index of cam profile data
        8272 = 3600000 (Name=CURVE_X_FACTOR+0)  // FB0 CURVE Multiplication factor for input interval
        8280 = 324000 (Name=CURVE_Y_FACTOR+0)  // FB0 CURVE Multiplication factor for output interval
        8192 = 2 (Name=CURVE_MODE+0)  // FB0 CURVE Mode
      ARITH 0:
        3584 = 0 (Name=ARITH_MODE+0)  // FB0 ARITH Mode
        3592 = CURVE_VALUE_I4+0 (Name=ARITH_IN1_PARID+0)  // FB0 ARITH Parameter ID of input1
        3600 = VAR_I4_1+0 (Name=ARITH_IN2_PARID+0)  // FB0 ARITH Parameter ID of input2
        3632 = 1 (Name=ARITH_K1+0)  // FB0 ARITH Multiplication factor1
        3640 = 1 (Name=ARITH_K2+0)  // FB0 ARITH Multiplication factor2
        3584 = 1 (Name=ARITH_MODE+0)  // FB0 ARITH Mode
      CURVE 1:
        8193 = 0 (Name=CURVE_MODE+1)  // FB1 FB CURVE: Mode
        8201 = ARITH_VALUE_I4+0 (Name=CURVE_IN_PARID+1)  // FB1 FB CURVE: Parameter ID of input
        8209 = 65535 (Name=CURVE_AUT_DATA_INDEX+1)  // FB1 FB CURVE: Index of cam profile data
        8273 = 36000 (Name=CURVE_X_FACTOR+1)  // FB1 FB CURVE: Multiplication factor for input interval
        8281 = 36000 (Name=CURVE_Y_FACTOR+1)  // FB1 FB CURVE: Multiplication factor for output interval
        8193 = 2 (Name=CURVE_MODE+1)  // FB1 FB CURVE: Mode
      CURVE 3:
        8195 = 0 (Name=CURVE_MODE+3)  // FB3 FB CURVE: Mode
        8203 = VAR_I4_3+0 (Name=CURVE_IN_PARID+3)  // FB3 FB CURVE: Parameter ID of input
        8211 = 65535 (Name=CURVE_AUT_DATA_INDEX+3)  // FB3 FB CURVE: Index of cam profile data
        8275 = 3600000 (Name=CURVE_X_FACTOR+3)  // FB3 FB CURVE: Multiplication factor for input interval
        8283 = 324000 (Name=CURVE_Y_FACTOR+3)  // FB3 FB CURVE: Multiplication factor for output interval
        8195 = 2 (Name=CURVE_MODE+3)  // FB3 FB CURVE: Mode
      CURVE 4:
        8196 = 0 (Name=CURVE_MODE+4)  // FB4 FB CURVE: Mode
        8204 = CURVE_VALUE_I4+3 (Name=CURVE_IN_PARID+4)  // FB4 FB CURVE: Parameter ID of input
        8212 = 65535 (Name=CURVE_AUT_DATA_INDEX+4)  // FB4 FB CURVE: Index of cam profile data
        8276 = 36000 (Name=CURVE_X_FACTOR+4)  // FB4 FB CURVE: Multiplication factor for input interval
        8284 = 36000 (Name=CURVE_Y_FACTOR+4)  // FB4 FB CURVE: Multiplication factor for output interval
        8196 = 2 (Name=CURVE_MODE+4)  // FB4 FB CURVE: Mode
      CURVE 5:
        8197 = 0 (Name=CURVE_MODE+5)  // FB5 FB CURVE: Mode
        8205 = S_SET_VAX1 (Name=CURVE_IN_PARID+5)  // FB5 FB CURVE: Parameter ID of input
        8213 = 65535 (Name=CURVE_AUT_DATA_INDEX+5)  // FB5 FB CURVE: Index of cam data
        8277 = 36000 (Name=CURVE_X_FACTOR+5)  // FB5 FB CURVE: Multiplication factor for input interval
        8285 = 36000 (Name=CURVE_Y_FACTOR+5)  // FB5 FB CURVE: Multiplication factor for output interval
        8197 = 2 (Name=CURVE_MODE+5)  // FB5 FB CURVE: Mode
```

### Data object Logical/30_MC/AxisTable/VirtualTables/gVirtualIn (Vax) - ACP10: Virtual Axis data object.

- gVirtIn.vax (not shown)

### Package Logical/30_MC/AxisTable/PwrSupplyTables - gPwrAxisobj

### Data object Logical/30_MC/AxisTable/PwrSupplyTables/gPwrPr (Apt)

#### gPwrAxisa.apt
```
AcoposParameterTable:
  Root Parameters:
    COMMON:
      80 = 1 (Name=PHASE_MON_IGNORE)  // Power mains: Ignore phase failure
      368 = 0 (Name=UVLIM_MODE)  // CTRL DC bus: Limiter: Mode
      351 = 0 (Name=ERRESP_UDC_POWERFAIL)  // Power mains: Error response
      390 = 400 (Name=UDC_NOMINAL, Unit=V)  // CTRL DC bus: Nominal voltage
    Declaration:
      777 = CMP_MODE+0 (Name=FUNCTION_BLOCK_CREATE)  // Function block: Create a FB instance
      777 = CMP_MODE+1 (Name=FUNCTION_BLOCK_CREATE)  // Function block: Create a FB instance
      777 = CMP_MODE+2 (Name=FUNCTION_BLOCK_CREATE)  // Function block: Create a FB instance
      777 = BIT_MODE+0 (Name=FUNCTION_BLOCK_CREATE)  // Function block: Create a FB instance
      777 = ARITH_MODE+5 (Name=FUNCTION_BLOCK_CREATE)  // Function block: Create a FB instance
      777 = VAR_R4_0+0 (Name=FUNCTION_BLOCK_CREATE)  // Function block: Create a FB instance
    Bleeder:
      345 = 750 (Name=UDC_BLEEDER_ON, Unit=V)  // CTRL DC bus: Limiter: Switch on threshold
      10 = 33 (Name=R_BLEEDER_EXT, Unit=Ohm)  // Bleeder: External: Resistance
      11 = 670 (Name=TEMP_MAX_BLEEDER_EXT, Unit=°C)  // Bleeder: External: Limit temperature
      12 = 0.852 (Name=RTH_BLEEDER_AMB_EXT, Unit=K/W)  // Bleeder: External: Thermal resistance
      13 = 22.6 (Name=CTH_BLEEDER_EXT, Unit=Ws/K)  // Bleeder: External: Thermal capacity
      398 = 1 (Name=BLEEDER_SELECTOR_EXT)  // Bleeder: Selector
      6689 = 0 (Name=CMP_MODE+1)  // FB0 CMP mode
      6657 = TEMP_BLEEDER (Name=CMP_IN_PARID+1)  // FB0 CMP parameter ID of input
      6665 = 620 (Name=CMP_THRESHOLD+1)  // FB0 CMP threshold
      6673 = 0 (Name=CMP_WINDOW+1)  // FB0 CMP window
      6681 = 0 (Name=CMP_HYSTERESIS+1)  // FB0 CMP hysteresis window
      6689 = 6 (Name=CMP_MODE+1)  // FB0 CMP mode
    POWER FAIL MANAGEMENT:
      6688 = 0 (Name=CMP_MODE+0)  // FB0 CMP mode
      6656 = UDC_ACT (Name=CMP_IN_PARID+0)  // FB0 CMP parameter ID of input
      6664 = 480 (Name=CMP_THRESHOLD+0)  // FB0 CMP threshold
      6672 = 0 (Name=CMP_WINDOW+0)  // FB0 CMP window
      6680 = 0 (Name=CMP_HYSTERESIS+0)  // FB0 CMP hysteresis window
      6688 = 3 (Name=CMP_MODE+0)  // FB0 CMP mode
    SUPPLY VOLTAGE CALCULATION  // Voltage Monitor
      4128 = 1.414 (Name=VAR_R4_0+0)  // FB0 FB VAR: Variable0 R4
      3589 = 0 (Name=ARITH_MODE+5)  // FB5 FB ARITH: Mode
      3597 = UDC_ACT (Name=ARITH_IN1_PARID+5)  // FB5 FB ARITH: Parameter ID of input1
      3605 = VAR_R4_0+0 (Name=ARITH_IN2_PARID+5)  // FB5 FB ARITH: Parameter ID of input2
      3589 = 5 (Name=ARITH_MODE+5)  // FB5 FB ARITH: Mode
    SUPPLY VOLTAGE CHECK  // Voltage Monitor
      6690 = 0 (Name=CMP_MODE+2)  // FB0 CMP mode
      6658 = ARITH_VALUE_R4+5 (Name=CMP_IN_PARID+2)  // FB0 CMP parameter ID of input
      6666 = 360 (Name=CMP_THRESHOLD+2)  // FB0 CMP threshold
      6690 = 3 (Name=CMP_MODE+2)  // FB0 CMP mode
    POWER SUPPLY ERROR MUX:
      12800 = 0 (Name=BIT_MODE+0)  // FB0 BIT Mode
      12808 = 16 (Name=BIT_A1+0)  // FB0 BIT Operand a1 - Gc_PhaseMonitorError
      12816 = 1 (Name=BIT_A2+0)  // FB0 BIT Operand a2 - Gc_DcBusUndervoltageError
      12824 = 1 (Name=BIT_A3+0)  // FB0 FB BIT: Operand a3 - Gc_BleederError
      12832 = 1 (Name=BIT_A4+0)  // FB0 FB BIT: Operand a4 - Gc_PowerSupplyVoltageMonitor
      12872 = 0 (Name=BIT_B1+0)  // FB0 BIT Operand b1
      12880 = 1 (Name=BIT_B2+0)  // FB0 BIT Operand b2
      12888 = 0 (Name=BIT_B3+0)  // FB0 FB BIT: Operand b3
      12896 = 2 (Name=BIT_B4+0)  // FB0 FB BIT: Operand b4 - Voltage Monitor
      12936 = STAT_PHASE_MON (Name=BIT_IN1_PARID+0)  // FB0 BIT Parameter ID of input1
      12944 = CMP_VALUE+0 (Name=BIT_IN2_PARID+0)  // FB0 BIT Parameter ID of input2
      12952 = CMP_VALUE+1 (Name=BIT_IN3_PARID+0)  // FB0 FB BIT: Parameter ID of input3
      12960 = CMP_VALUE+2 (Name=BIT_IN4_PARID+0)  // FB0 FB BIT: Parameter ID of input4
      12800 = 4 (Name=BIT_MODE+0)  // FB0 BIT Mode
```

### Data object Logical/30_MC/AxisTable/PwrSupplyTables/gPwrIn (Ax)

#### gPwrAxisi.ax
```
InitParameter (Version=2.51.0, NcSwId=ACP10)
  ACP10AXIS_typ:
    dig_in:
      level:
        reference = ncACTIV_HI
        pos_hw_end = ncACTIV_HI
        neg_hw_end = ncACTIV_HI
        trigger1 = ncACTIV_HI
        trigger2 = ncACTIV_HI
    encoder_if:
      parameter:
        count_dir = ncSTANDARD
        scaling:
          load:
            units = 36000
            rev_motor = 1
    limit:
      parameter:
        v_pos = 10000.0
        v_neg = 10000.0
        a1_pos = 50000.0
        a2_pos = 50000.0
        a1_neg = 50000.0
        a2_neg = 50000.0
        t_jolt = 0.0
        t_in_pos = 0.0
        pos_sw_end = 8388607
        neg_sw_end = -8388608
        ds_warning = 500.0
        ds_stop = 1000.0
        a_stop = 1.0e+30
        dv_stop = 0.0
        dv_stop_mode = ncOFF
    controller:
      mode = ncPOSITION
      position:
        kv = 50.0
        tn = 0.0
        t_predict = 0.0004
        t_total = 0.0004
        p_max = 1.0e+30
        i_max = 0.0
      speed:
        kv = 2.0
        tn = 0.0
        t_filter = 0.0
        isq_filter1:
          type = ncOFF
          a0 = 0.0
          a1 = 0.0
          b0 = 0.0
          b1 = 0.0
          b2 = 0.0
          c0_par_id = 0
          c1_par_id = 0
        isq_filter2:
          type = ncOFF
          a0 = 0.0
          a1 = 0.0
          b0 = 0.0
          b1 = 0.0
          b2 = 0.0
          c0_par_id = 0
          c1_par_id = 0
        isq_filter3:
          type = ncOFF
          a0 = 0.0
          a1 = 0.0
          b0 = 0.0
          b1 = 0.0
          b2 = 0.0
          c0_par_id = 0
          c1_par_id = 0
      uf:
        type = ncLINEAR
        auto_config = ncMOTOR_PAR
        u0 = 0.0
        un = 0.0
        fn = 50.0
        k_f_slip = 0.0
      ff:
        torque_load = 0.0
        torque_pos = 0.0
        torque_neg = 0.0
        kv_torque = 0.0
        inertia = 0.0
        t_filter_a = 0.0
    move:
      stop:
        parameter[0]:
          decel_ramp = ncA_LIMIT
          controller = ncON
        parameter[1]:
          decel_ramp = ncA_LIMIT
          controller = ncON
        parameter[2]:
          decel_ramp = ncA_LIMIT
          controller = ncON
        parameter[3]:
          decel_ramp = ncA_LIMIT
          controller = ncON
        quickstop:
          decel_ramp = ncA_LIMIT
        drive_error:
          decel_ramp = ncA_LIMIT
      homing:
        parameter:
          s = 0
          v_switch = 5000.0
          v_trigger = 500.0
          a = 50000.0
          mode = ncDIRECT
          edge_sw = ncPOSITIVE
          start_dir = ncPOSITIVE
          trigg_dir = ncPOSITIVE
          ref_pulse = ncOFF
          fix_dir = ncOFF
          tr_s_block = 0.0
          torque_lim = 0.0
          ds_block = 0.0
          ds_stop = 0.0
      basis:
        parameter:
          v_pos = 5000.0
          v_neg = 5000.0
          a1_pos = 50000.0
          a2_pos = 50000.0
          a1_neg = 50000.0
          a2_neg = 50000.0
    message:
      text:
        parameter:
          format = ncBREAK + ncZERO
          columns = 80
          data_modul = acp10etxen
```

### Package Logical/30_MC/AxisTable/RealTablesNoBrake - gMasterAxobj

### Data object Logical/30_MC/AxisTable/RealTablesNoBrake/gRealNoBrake (Apt)

#### gRealNoBrake.apt
```
AcoposParameterTable:
  Root Parameters:
    COMMON_INITIALIZATION:
      90 = 0 (Name=BRAKE_MODE)  // Disable Motor holding brake automatic management
      128 = 1 (Name=SGEN_SW_END_IGNORE)  // Limit values: Ignore SW end positions
      368 = 0 (Name=UVLIM_MODE)  // CTRL DC bus: Limiter: Mode (DcBus Alarm Off)
      390 = 400 (Name=UDC_NOMINAL, Unit=V)  // CTRL DC bus: Nominal voltage
      351 = 0 (Name=ERRESP_UDC_POWERFAIL)  // Power mains: Error response
      347 = 10000 (Name=F_SWITCH, Unit=cps)  // Power stage: Switch frequency
      602 = 2 (Name=MA1_CYCLIC_IPL_MODE)  // Network coupling: Interpolation mode for cyclic position master1
    Torque And Lag Error Control:
      Declarations:
        777 = CMP_MODE+0 (Name=FUNCTION_BLOCK_CREATE)  // Function block: Create a FB instance
        777 = CMP_MODE+1 (Name=FUNCTION_BLOCK_CREATE)  // Function block: Create a FB instance
        777 = VAR_I4_0+0 (Name=FUNCTION_BLOCK_CREATE)  // Function block: Create a FB instance
        777 = BIT_MODE+0 (Name=FUNCTION_BLOCK_CREATE)  // Function block: Create a FB instance
      Torque Control:
        6688 = 0 (Name=CMP_MODE+0)  // FB0 CMP mode : <>
        6656 = TORQUE_ACT (Name=CMP_IN_PARID+0)  // FB0 CMP parameter ID of input
        6664 = 0 (Name=CMP_THRESHOLD+0)  // FB0 CMP threshold
        6672 = 0 (Name=CMP_WINDOW+0)  // FB0 CMP window - This value has to be written on grey code = Limit Value
        6680 = 0 (Name=CMP_HYSTERESIS+0)  // FB0 CMP hysteresis window
        6688 = 5 (Name=CMP_MODE+0)  // FB0 CMP mode : <>
      Lag Error Control:
        6689 = 0 (Name=CMP_MODE+1)  // FB0 CMP mode
        6657 = PCTRL_LAG_ERROR (Name=CMP_IN_PARID+1)  // FB0 CMP parameter ID of input
        6665 = 0 (Name=CMP_THRESHOLD+1)  // FB0 CMP threshold
        6673 = 1e6 (Name=CMP_WINDOW+1)  // FB0 CMP window - This value has to be written on grey code = Limit Value
        6681 = 0 (Name=CMP_HYSTERESIS+1)  // FB0 CMP hysteresis window
        6689 = 5 (Name=CMP_MODE+1)  // FB0 CMP mode
      BIT:
        12800 = 0 (Name=BIT_MODE+0)  // FB0 BIT Mode
        12808 = 1 (Name=BIT_A1+0)  // FB0 BIT Operand a1
        12816 = 1 (Name=BIT_A2+0)  // FB0 BIT Operand a2
        12824 = 8 (Name=BIT_A3+0)  // FB0 FB BIT: Operand a3
        12872 = 0 (Name=BIT_B1+0)  // FB0 BIT Operand b1
        12880 = 1 (Name=BIT_B2+0)  // FB0 BIT Operand b2
        12888 = 0 (Name=BIT_B3+0)  // FB0 FB BIT: Operand b3
        12936 = CMP_VALUE+0 (Name=BIT_IN1_PARID+0)  // FB0 BIT Parameter ID of input1
        12944 = CMP_VALUE+1 (Name=BIT_IN2_PARID+0)  // FB0 BIT Parameter ID of input2
        12952 = STATUS_BITS (Name=BIT_IN3_PARID+0)  // FB0 FB BIT: Parameter ID of input3
        12800 = 4 (Name=BIT_MODE+0)  // FB0 BIT Mode
```

### Data object Logical/30_MC/AxisTable/RealTablesNoBrake/gRealNoBrakeIn (Ax)

#### gRealNoBrake.ax
```
InitParameter (Version=2.51.0, NcSwId=ACP10)
  ACP10AXIS_typ:
    dig_in:
      level:
        reference = ncACTIV_HI
        pos_hw_end = ncACTIV_HI
        neg_hw_end = ncACTIV_HI
        trigger1 = ncACTIV_HI
        trigger2 = ncACTIV_HI
    encoder_if:
      parameter:
        count_dir = ncSTANDARD
        scaling:
          load:
            units = 1296000
            rev_motor = 27
    limit:
      parameter:
        v_pos = 1800000.0
        v_neg = 1800000.0
        a1_pos = 5000000.0
        a2_pos = 5000000.0
        a1_neg = 5000000.0
        a2_neg = 5000000.0
        t_jolt = 0.0
        t_in_pos = 0.0
        pos_sw_end = 838860700
        neg_sw_end = -838860800
        ds_warning = 1.0e+32
        ds_stop = 1.0e+32
        a_stop = 1.0e+30
        dv_stop = 1.0e+32
        dv_stop_mode = ncDV_STOP_INIT
    controller:
      mode = ncPOSITION
      position:
        kv = 1.0
        tn = 0.0
        t_predict = 0.0004
        t_total = 0.0004
        p_max = 1.0e+30
        i_max = 50000.0
      speed:
        kv = 1.0
        tn = 0.0
        t_filter = 0.0
        isq_filter1:
          type = ncOFF
          a0 = 0.0
          a1 = 0.0
          b0 = 0.0
          b1 = 0.0
          b2 = 0.0
          c0_par_id = 0
          c1_par_id = 0
        isq_filter2:
          type = ncOFF
          a0 = 0.0
          a1 = 0.0
          b0 = 0.0
          b1 = 0.0
          b2 = 0.0
          c0_par_id = 0
          c1_par_id = 0
        isq_filter3:
          type = ncOFF
          a0 = 0.0
          a1 = 0.0
          b0 = 0.0
          b1 = 0.0
          b2 = 0.0
          c0_par_id = 0
          c1_par_id = 0
      uf:
        type = ncLINEAR
        auto_config = ncMOTOR_PAR
        u0 = 0.0
        un = 0.0
        fn = 50.0
        k_f_slip = 0.0
      ff:
        torque_load = 0.0
        torque_pos = 0.0
        torque_neg = 0.0
        kv_torque = 0.0
        inertia = 0.0
        t_filter_a = 0.0
    move:
      stop:
        parameter[0]:
          decel_ramp = ncA_LIMIT
          controller = ncON
        parameter[1]:
          decel_ramp = ncA_LIMIT
          controller = ncON
        parameter[2]:
          decel_ramp = ncA_LIMIT
          controller = ncON
        parameter[3]:
          decel_ramp = ncA_LIMIT
          controller = ncON
        quickstop:
          decel_ramp = ncA_LIMIT
        drive_error:
          decel_ramp = ncA_LIMIT
      homing:
        parameter:
          s = 6960
          v_switch = 5000.0
          v_trigger = 500.0
          a = 50000.0
          mode = ncHOME_OFFSET
          edge_sw = ncPOSITIVE
          start_dir = ncPOSITIVE
          trigg_dir = ncPOSITIVE
          ref_pulse = ncOFF
          fix_dir = ncOFF
          tr_s_block = 0.0
          torque_lim = 0.0
          ds_block = 0.0
          ds_stop = 0.0
      basis:
        parameter:
          v_pos = 10000.0
          v_neg = 10000.0
          a1_pos = 80000.0
          a2_pos = 400000.0
          a1_neg = 80000.0
          a2_neg = 400000.0
    message:
      text:
        parameter:
          format = ncBREAK + ncZERO
          columns = 80
          data_modul = acp10etxen
```

### Package Logical/30_MC/AxisTable/RealTablesWithBrake - gMasterAxobj

### Data object Logical/30_MC/AxisTable/RealTablesWithBrake/gRealWithBrake (Apt)

#### gRealBrake.apt
```
AcoposParameterTable:
  Root Parameters:
    COMMON_INITIALIZATION:
      128 = 1 (Name=SGEN_SW_END_IGNORE)  // Limit values: Ignore SW end positions
      368 = 0 (Name=UVLIM_MODE)  // CTRL DC bus: Limiter: Mode (DcBus Alarm Off)
      390 = 400 (Name=UDC_NOMINAL, Unit=V)  // CTRL DC bus: Nominal voltage
      351 = 0 (Name=ERRESP_UDC_POWERFAIL)  // Power mains: Error response
      347 = 10000 (Name=F_SWITCH, Unit=cps)  // Power stage: Switch frequency
      602 = 2 (Name=MA1_CYCLIC_IPL_MODE)  // Network coupling: Interpolation mode for cyclic position master1
    Torque And Lag Error Control:
      Declarations:
        777 = CMP_MODE+0 (Name=FUNCTION_BLOCK_CREATE)  // Function block: Create a FB instance
        777 = CMP_MODE+1 (Name=FUNCTION_BLOCK_CREATE)  // Function block: Create a FB instance
        777 = VAR_I4_0+0 (Name=FUNCTION_BLOCK_CREATE)  // Function block: Create a FB instance
        777 = BIT_MODE+0 (Name=FUNCTION_BLOCK_CREATE)  // Function block: Create a FB instance
      Torque Control:
        6688 = 0 (Name=CMP_MODE+0)  // FB0 CMP mode : <>
        6656 = TORQUE_ACT (Name=CMP_IN_PARID+0)  // FB0 CMP parameter ID of input
        6664 = 0 (Name=CMP_THRESHOLD+0)  // FB0 CMP threshold
        6672 = 0 (Name=CMP_WINDOW+0)  // FB0 CMP window - This value has to be written on grey code = Limit Value
        6680 = 0 (Name=CMP_HYSTERESIS+0)  // FB0 CMP hysteresis window
        6688 = 5 (Name=CMP_MODE+0)  // FB0 CMP mode : <>
      Lag Error Control:
        6689 = 0 (Name=CMP_MODE+1)  // FB0 CMP mode
        6657 = PCTRL_LAG_ERROR (Name=CMP_IN_PARID+1)  // FB0 CMP parameter ID of input
        6665 = 0 (Name=CMP_THRESHOLD+1)  // FB0 CMP threshold
        6673 = 1e6 (Name=CMP_WINDOW+1)  // FB0 CMP window - This value has to be written on grey code = Limit Value
        6681 = 0 (Name=CMP_HYSTERESIS+1)  // FB0 CMP hysteresis window
        6689 = 5 (Name=CMP_MODE+1)  // FB0 CMP mode
      BIT:
        12800 = 0 (Name=BIT_MODE+0)  // FB0 BIT Mode
        12808 = 1 (Name=BIT_A1+0)  // FB0 BIT Operand a1
        12816 = 1 (Name=BIT_A2+0)  // FB0 BIT Operand a2
        12824 = 8 (Name=BIT_A3+0)  // FB0 FB BIT: Operand a3
        12872 = 0 (Name=BIT_B1+0)  // FB0 BIT Operand b1
        12880 = 1 (Name=BIT_B2+0)  // FB0 BIT Operand b2
        12888 = 0 (Name=BIT_B3+0)  // FB0 FB BIT: Operand b3
        12936 = CMP_VALUE+0 (Name=BIT_IN1_PARID+0)  // FB0 BIT Parameter ID of input1
        12944 = CMP_VALUE+1 (Name=BIT_IN2_PARID+0)  // FB0 BIT Parameter ID of input2
        12952 = STATUS_BITS (Name=BIT_IN3_PARID+0)  // FB0 FB BIT: Parameter ID of input3
        12800 = 4 (Name=BIT_MODE+0)  // FB0 BIT Mode
```

### Data object Logical/30_MC/AxisTable/RealTablesWithBrake/gRealWithBrakeIn (Ax)

#### gRealBrake.ax
```
InitParameter (Version=3.17.2, NcSwId=ACP10)
  ACP10AXIS_typ:
    dig_in:
      level:
        reference = ncACTIV_HI
        pos_hw_end = ncACTIV_HI
        neg_hw_end = ncACTIV_HI
        trigger1 = ncACTIV_HI
        trigger2 = ncACTIV_HI
    encoder_if:
      parameter:
        count_dir = ncSTANDARD
        scaling:
          load:
            units = 1296000
            rev_motor = 27
    limit:
      parameter:
        v_pos = 1800000.0
        v_neg = 1800000.0
        a1_pos = 5000000.0
        a2_pos = 5000000.0
        a1_neg = 5000000.0
        a2_neg = 5000000.0
        t_jolt = 0.0
        t_in_pos = 0.0
        pos_sw_end = 838860700
        neg_sw_end = -838860800
        ds_warning = 1.0e+32
        ds_stop = 1.0e+32
        a_stop = 1.0e+30
        dv_stop = 1.0e+32
        dv_stop_mode = ncDV_STOP_INIT
    controller:
      mode = ncPOSITION
      position:
        kv = 1.0
        tn = 0.0
        t_predict = 0.0004
        t_total = 0.0004
        p_max = 1.0e+30
        i_max = 1.0e+30
      speed:
        kv = 1.0
        tn = 0.0
        t_filter = 0.0
        isq_filter1:
          type = ncOFF
          a0 = 0.0
          a1 = 0.0
          b0 = 0.0
          b1 = 0.0
          b2 = 0.0
          c0_par_id = 0
          c1_par_id = 0
        isq_filter2:
          type = ncOFF
          a0 = 0.0
          a1 = 0.0
          b0 = 0.0
          b1 = 0.0
          b2 = 0.0
          c0_par_id = 0
          c1_par_id = 0
        isq_filter3:
          type = ncOFF
          a0 = 0.0
          a1 = 0.0
          b0 = 0.0
          b1 = 0.0
          b2 = 0.0
          c0_par_id = 0
          c1_par_id = 0
      uf:
        type = ncLINEAR
        auto_config = ncMOTOR_PAR
        u0 = 0.0
        un = 0.0
        fn = 50.0
        k_f_slip = 0.0
      ff:
        torque_load = 0.0
        torque_pos = 0.0
        torque_neg = 0.0
        kv_torque = 0.0
        inertia = 0.0
        t_filter_a = 0.0
    move:
      stop:
        parameter[0]:
          decel_ramp = ncA_LIMIT
          controller = ncON
        parameter[1]:
          decel_ramp = ncA_LIMIT
          controller = ncON
        parameter[2]:
          decel_ramp = ncA_LIMIT
          controller = ncON
        parameter[3]:
          decel_ramp = ncA_LIMIT
          controller = ncON
        quickstop:
          decel_ramp = ncA_LIMIT
        drive_error:
          decel_ramp = ncA_LIMIT
      homing:
        parameter:
          s = 6960
          v_switch = 5000.0
          v_trigger = 500.0
          a = 50000.0
          mode = ncHOME_OFFSET
          edge_sw = ncPOSITIVE
          start_dir = ncPOSITIVE
          trigg_dir = ncPOSITIVE
          ref_pulse = ncOFF
          fix_dir = ncOFF
          tr_s_block = 0.0
          torque_lim = 0.0
          ds_block = 0.0
          ds_stop = 0.0
      basis:
        parameter:
          v_pos = 10000.0
          v_neg = 10000.0
          a1_pos = 80000.0
          a2_pos = 400000.0
          a1_neg = 80000.0
          a2_neg = 400000.0
    message:
      text:
        parameter:
          format = ncBREAK + ncZERO
          columns = 80
          data_modul = acp10etxen
```

### Package Logical/30_MC/AxisTable/RealTablesOnlyVelocity - gMasterAxobj

### Data object Logical/30_MC/AxisTable/RealTablesOnlyVelocity/gRealVelAsync (Apt)

#### gRealVelAsync.apt
```
AcoposParameterTable:
  Root Parameters:
    COMMON_INITIALIZATION:
      128 = 1 (Name=SGEN_SW_END_IGNORE)  // Limit values: Ignore SW end positions
      368 = 0 (Name=UVLIM_MODE)  // CTRL DC bus: Limiter: Mode (DcBus Alarm Off)
      390 = 400 (Name=UDC_NOMINAL, Unit=V)  // CTRL DC bus: Nominal voltage
      347 = 5000 (Name=F_SWITCH, Unit=cps)  // Power stage: Switch frequency
      351 = 0 (Name=ERRESP_UDC_POWERFAIL)  // Power mains: Error response
      602 = 2 (Name=MA1_CYCLIC_IPL_MODE)  // Network coupling: Interpolation mode for cyclic position master1
      230 = PCTRL_S_SET (Name=PCTRL_S_ACT_PARID, Disabled=FALSE)  // CTRL Position controller: Actual encoder position parameter ID - The Loop Is Open
      86 = 259 (Name=CMD_BRAKE, Disabled=TRUE)  // Motor holding brake: Command - Per Sbloccare Freno 259 - Per bloccare 258
    Torque And Lag Error Control:
      Declarations:
        777 = CMP_MODE+0 (Name=FUNCTION_BLOCK_CREATE)  // Function block: Create a FB instance
        777 = CMP_MODE+1 (Name=FUNCTION_BLOCK_CREATE)  // Function block: Create a FB instance
        777 = VAR_I4_0+0 (Name=FUNCTION_BLOCK_CREATE)  // Function block: Create a FB instance
        777 = BIT_MODE+0 (Name=FUNCTION_BLOCK_CREATE)  // Function block: Create a FB instance
      Torque Control:
        6688 = 0 (Name=CMP_MODE+0)  // FB0 CMP mode : <>
        6656 = TORQUE_ACT (Name=CMP_IN_PARID+0)  // FB0 CMP parameter ID of input
        6664 = 0 (Name=CMP_THRESHOLD+0)  // FB0 CMP threshold
        6672 = 0 (Name=CMP_WINDOW+0)  // FB0 CMP window - This value has to be written on grey code = Limit Value
        6680 = 0 (Name=CMP_HYSTERESIS+0)  // FB0 CMP hysteresis window
        6688 = 5 (Name=CMP_MODE+0)  // FB0 CMP mode : <>
      Lag Error Control:
        6689 = 0 (Name=CMP_MODE+1)  // FB0 CMP mode
        6657 = PCTRL_LAG_ERROR (Name=CMP_IN_PARID+1)  // FB0 CMP parameter ID of input
        6665 = 0 (Name=CMP_THRESHOLD+1)  // FB0 CMP threshold
        6673 = 1e6 (Name=CMP_WINDOW+1)  // FB0 CMP window - This value has to be written on grey code = Limit Value
        6681 = 0 (Name=CMP_HYSTERESIS+1)  // FB0 CMP hysteresis window
        6689 = 5 (Name=CMP_MODE+1)  // FB0 CMP mode
      BIT:
        12800 = 0 (Name=BIT_MODE+0)  // FB0 BIT Mode
        12808 = 1 (Name=BIT_A1+0)  // FB0 BIT Operand a1
        12816 = 1 (Name=BIT_A2+0)  // FB0 BIT Operand a2
        12872 = 0 (Name=BIT_B1+0)  // FB0 BIT Operand b1
        12880 = 1 (Name=BIT_B2+0)  // FB0 BIT Operand b2
        12936 = CMP_VALUE+0 (Name=BIT_IN1_PARID+0)  // FB0 BIT Parameter ID of input1
        12944 = CMP_VALUE+1 (Name=BIT_IN2_PARID+0)  // FB0 BIT Parameter ID of input2
        12800 = 4 (Name=BIT_MODE+0)  // FB0 BIT Mode
```

### Data object Logical/30_MC/AxisTable/RealTablesOnlyVelocity/gRealVelSync (Apt)

#### gRealVelSync.apt
```
AcoposParameterTable:
  Root Parameters:
    COMMON_INITIALIZATION:
      128 = 1 (Name=SGEN_SW_END_IGNORE)  // Limit values: Ignore SW end positions
      368 = 0 (Name=UVLIM_MODE)  // CTRL DC bus: Limiter: Mode (DcBus Alarm Off)
      390 = 400 (Name=UDC_NOMINAL, Unit=V)  // CTRL DC bus: Nominal voltage
      347 = 5000 (Name=F_SWITCH, Unit=cps)  // Power stage: Switch frequency
      351 = 0 (Name=ERRESP_UDC_POWERFAIL)  // Power mains: Error response
      602 = 2 (Name=MA1_CYCLIC_IPL_MODE)  // Network coupling: Interpolation mode for cyclic position master1
      230 = ENCOD0_S_ACT (Name=PCTRL_S_ACT_PARID)  // CTRL Position controller: Actual encoder position parameter ID - The Loop Is Open
      90 = 0 (Name=BRAKE_MODE, Disabled=FALSE)  // Motor holding brake: Mode
    Torque And Lag Error Control:
      Declarations:
        777 = CMP_MODE+0 (Name=FUNCTION_BLOCK_CREATE)  // Function block: Create a FB instance
        777 = CMP_MODE+1 (Name=FUNCTION_BLOCK_CREATE)  // Function block: Create a FB instance
        777 = VAR_I4_0+0 (Name=FUNCTION_BLOCK_CREATE)  // Function block: Create a FB instance
        777 = VAR_R4_0+0 (Name=FUNCTION_BLOCK_CREATE)  // Function block: Create a FB instance
        777 = BIT_MODE+0 (Name=FUNCTION_BLOCK_CREATE)  // Function block: Create a FB instance
      Torque Control:
        6688 = 0 (Name=CMP_MODE+0)  // FB0 CMP mode : <>
        6656 = TORQUE_ACT (Name=CMP_IN_PARID+0)  // FB0 CMP parameter ID of input
        6664 = 0 (Name=CMP_THRESHOLD+0)  // FB0 CMP threshold
        6672 = 0 (Name=CMP_WINDOW+0)  // FB0 CMP window - This value has to be written on grey code = Limit Value
        6680 = 0 (Name=CMP_HYSTERESIS+0)  // FB0 CMP hysteresis window
        6688 = 5 (Name=CMP_MODE+0)  // FB0 CMP mode : <>
      Lag Error Control:
        6689 = 0 (Name=CMP_MODE+1)  // FB0 CMP mode
        6657 = PCTRL_LAG_ERROR (Name=CMP_IN_PARID+1)  // FB0 CMP parameter ID of input
        6665 = 0 (Name=CMP_THRESHOLD+1)  // FB0 CMP threshold
        6673 = 1e6 (Name=CMP_WINDOW+1)  // FB0 CMP window - This value has to be written on grey code = Limit Value
        6681 = 0 (Name=CMP_HYSTERESIS+1)  // FB0 CMP hysteresis window
        6689 = 5 (Name=CMP_MODE+1)  // FB0 CMP mode
      BIT:
        12800 = 0 (Name=BIT_MODE+0)  // FB0 BIT Mode
        12808 = 1 (Name=BIT_A1+0)  // FB0 BIT Operand a1
        12816 = 1 (Name=BIT_A2+0)  // FB0 BIT Operand a2
        12872 = 0 (Name=BIT_B1+0)  // FB0 BIT Operand b1
        12880 = 1 (Name=BIT_B2+0)  // FB0 BIT Operand b2
        12936 = CMP_VALUE+0 (Name=BIT_IN1_PARID+0)  // FB0 BIT Parameter ID of input1
        12944 = CMP_VALUE+1 (Name=BIT_IN2_PARID+0)  // FB0 BIT Parameter ID of input2
        12800 = 4 (Name=BIT_MODE+0)  // FB0 BIT Mode
    1320 = 1 (Name=ENCOD0_MODE)  // Virtual Encoder: Mode
    722 = ENCOD0_S_ACT (Name=VCTRL_S_ACT_PARID)  // CTRL Vector controller: Actual position parameter ID
    276 = 0 (Name=PHASING_MODE)  // Motor: Phasing: Mode
```

### Data object Logical/30_MC/AxisTable/RealTablesOnlyVelocity/gRealVelIn (Ax)

#### gRealVel.ax
```
InitParameter (Version=2.51.0, NcSwId=ACP10)
  ACP10AXIS_typ:
    dig_in:
      level:
        reference = ncACTIV_HI
        pos_hw_end = ncACTIV_HI
        neg_hw_end = ncACTIV_HI
        trigger1 = ncACTIV_HI
        trigger2 = ncACTIV_HI
    encoder_if:
      parameter:
        count_dir = ncSTANDARD
        scaling:
          load:
            units = 1296000
            rev_motor = 27
    limit:
      parameter:
        v_pos = 1800000.0
        v_neg = 1800000.0
        a1_pos = 5000000.0
        a2_pos = 5000000.0
        a1_neg = 5000000.0
        a2_neg = 5000000.0
        t_jolt = 0.0
        t_in_pos = 0.0
        pos_sw_end = 838860700
        neg_sw_end = -838860800
        ds_warning = 1.0e+32
        ds_stop = 1.0e+32
        a_stop = 1.0e+30
        dv_stop = 1.0e+32
        dv_stop_mode = ncDV_STOP_INIT
    controller:
      mode = ncPOSITION
      position:
        kv = 1.0
        tn = 0.0
        t_predict = 0.0004
        t_total = 0.0004
        p_max = 1.0e+30
        i_max = 1.0e+30
      speed:
        kv = 1.0
        tn = 0.0
        t_filter = 0.0
        isq_filter1:
          type = ncOFF
          a0 = 0.0
          a1 = 0.0
          b0 = 0.0
          b1 = 0.0
          b2 = 0.0
          c0_par_id = 0
          c1_par_id = 0
        isq_filter2:
          type = ncOFF
          a0 = 0.0
          a1 = 0.0
          b0 = 0.0
          b1 = 0.0
          b2 = 0.0
          c0_par_id = 0
          c1_par_id = 0
        isq_filter3:
          type = ncOFF
          a0 = 0.0
          a1 = 0.0
          b0 = 0.0
          b1 = 0.0
          b2 = 0.0
          c0_par_id = 0
          c1_par_id = 0
      uf:
        type = ncLINEAR
        auto_config = ncMOTOR_PAR
        u0 = 0.0
        un = 0.0
        fn = 50.0
        k_f_slip = 0.0
      ff:
        torque_load = 0.0
        torque_pos = 0.0
        torque_neg = 0.0
        kv_torque = 0.0
        inertia = 0.0
        t_filter_a = 0.0
    move:
      stop:
        parameter[0]:
          decel_ramp = ncA_LIMIT
          controller = ncON
        parameter[1]:
          decel_ramp = ncA_LIMIT
          controller = ncON
        parameter[2]:
          decel_ramp = ncA_LIMIT
          controller = ncON
        parameter[3]:
          decel_ramp = ncA_LIMIT
          controller = ncON
        quickstop:
          decel_ramp = ncA_LIMIT
        drive_error:
          decel_ramp = ncA_LIMIT
      homing:
        parameter:
          s = 6960
          v_switch = 5000.0
          v_trigger = 500.0
          a = 50000.0
          mode = ncHOME_OFFSET
          edge_sw = ncPOSITIVE
          start_dir = ncPOSITIVE
          trigg_dir = ncPOSITIVE
          ref_pulse = ncOFF
          fix_dir = ncOFF
          tr_s_block = 0.0
          torque_lim = 0.0
          ds_block = 0.0
          ds_stop = 0.0
      basis:
        parameter:
          v_pos = 10000.0
          v_neg = 10000.0
          a1_pos = 80000.0
          a2_pos = 400000.0
          a1_neg = 80000.0
          a2_neg = 400000.0
    message:
      text:
        parameter:
          format = ncBREAK + ncZERO
          columns = 80
          data_modul = acp10etxen
```

### Data object Logical/30_MC/AxisTable/EncoderEmulation/gEncEmulIn (Ax)

#### gEncEmul.ax
```
InitParameter (Version=3.14.3, NcSwId=ACP10)
  ACP10AXIS_typ:
    dig_in:
      level:
        reference = ncACTIV_HI
        pos_hw_end = ncACTIV_LO
        neg_hw_end = ncACTIV_LO
        trigger1 = ncACTIV_HI
        trigger2 = ncACTIV_LO + ncQUICKSTOP
    encoder_if:
      parameter:
        count_dir = ncSTANDARD
        scaling:
          load:
            units = 36000
            rev_motor = 1
    limit:
      parameter:
        v_pos = 1800000.0
        v_neg = 1800000.0
        a1_pos = 5000000.0
        a2_pos = 5000000.0
        a1_neg = 5000000.0
        a2_neg = 5000000.0
        t_jolt = 0
        t_in_pos = 0
        pos_sw_end = 2000000000
        neg_sw_end = -2000000000
        ds_warning = 500
        ds_stop = 1000
        a_stop = 1.0e30
        dv_stop = 0
        dv_stop_mode = ncOFF
    controller:
      mode = ncPOSITION
      position:
        kv = 50
        tn = 0
        t_predict = 0.0004
        t_total = 0.0004
        p_max = 10000
        i_max = 0
      speed:
        kv = 2.0
        tn = 0
        t_filter = 0.0
        isq_filter1:
          type = ncOFF
          a0 = 0.0
          a1 = 0.0
          b0 = 0.0
          b1 = 0.0
          b2 = 0.0
          c0_par_id = 0
          c1_par_id = 0
        isq_filter2:
          type = ncOFF
          a0 = 0.0
          a1 = 0.0
          b0 = 0.0
          b1 = 0.0
          b2 = 0.0
          c0_par_id = 0
          c1_par_id = 0
        isq_filter3:
          type = ncOFF
          a0 = 0.0
          a1 = 0.0
          b0 = 0.0
          b1 = 0.0
          b2 = 0.0
          c0_par_id = 0
          c1_par_id = 0
      uf:
        type = ncLINEAR
        auto_config = ncMOTOR_PAR
        u0 = 0
        un = 0
        fn = 50.0
        k_f_slip = 0
      ff:
        torque_load = 0.0
        torque_pos = 0.0
        torque_neg = 0.0
        kv_torque = 0.0
        inertia = 0.0
        t_filter_a = 0.0
    move:
      stop:
        parameter[0]:
          decel_ramp = ncA_LIMIT
          controller = ncON
        parameter[1]:
          decel_ramp = ncA_LIMIT
          controller = ncON
        parameter[2]:
          decel_ramp = ncA_LIMIT
          controller = ncON
        parameter[3]:
          decel_ramp = ncA_LIMIT
          controller = ncON
        quickstop:
          decel_ramp = ncA_LIMIT
        drive_error:
          decel_ramp = ncA_LIMIT
      homing:
        parameter:
          s = 0
          v_switch = 5000
          v_trigger = 500
          a = 50000
          mode = ncDIRECT
          edge_sw = ncPOSITIVE
          start_dir = ncPOSITIVE
          trigg_dir = ncPOSITIVE
          ref_pulse = ncOFF
          fix_dir = ncOFF
          tr_s_block = 0
          torque_lim = 0
          ds_block = 0
          ds_stop = 0
      basis:
        parameter:
          v_pos = 5000
          v_neg = 5000
          a1_pos = 50000
          a2_pos = 50000
          a1_neg = 50000
          a2_neg = 50000
    message:
      text:
        parameter:
          format = ncBREAK
          columns = 80
          data_modul
```

### Package Logical/30_MC/AxisTable/TempTables - gMasterAxobj

### Data object Logical/30_MC/AxisTable/TempTables/TempPha (Apt)

#### TempPha.apt
```
AcoposParameterTable:
  Root Parameters:
    Axis Parameter Identification, Synchronous Motor:
      Group  // General Parameters
        30 = 2 (Name=MOTOR_TYPE)  // Motor: Type
        1224 = 0 (Name=MOTOR_VENDOR_ID)  // Motor: Vendor ID
        652 = 0 (Name=MOTOR_ENCOD_ATTR)  // Motor: Encoder: Attribute
        Brake parameters:
          90 = 0 (Name=BRAKE_MODE)  // Disable Motor holding brake automatic management
          42 = 0 (Name=MOTOR_BRAKE_CURR_RATED, Unit=A)  // Motor holding brake: Rated current
          43 = 0 (Name=MOTOR_BRAKE_TORQ_RATED, Unit=Nm)  // Motor holding brake: Rated torque
          44 = 0 (Name=MOTOR_BRAKE_ON_TIME, Unit=s)  // Motor holding brake: Engaging delay
          45 = 0 (Name=MOTOR_BRAKE_OFF_TIME, Unit=s)  // Motor holding brake: Release delay
        31 = 0x0203 (Name=MOTOR_COMPATIBILITY)  // Motor: Software compatibility
        46 = 1 (Name=MOTOR_WIND_CONNECT)  // Motor: Winding connection
        62 = 0 (Name=MOTOR_INERTIA, Unit=kgm²)  // Motor: Moment of inertia
        849 = 0 (Name=MOTOR_TAU_THERM, Unit=s)  // Motor: Thermal time constant
      Thermo sensor parameters:
        64 = 0 (Name=MOTOR_TEMPSENS_PAR1)  // Temperature sensor: Parameter 1
        65 = 0 (Name=MOTOR_TEMPSENS_PAR2)  // Temperature sensor: Parameter 2
        66 = 0 (Name=MOTOR_TEMPSENS_PAR3)  // Temperature sensor: Parameter 3
        67 = 0 (Name=MOTOR_TEMPSENS_PAR4)  // Temperature sensor: Parameter 4
        68 = 0 (Name=MOTOR_TEMPSENS_PAR5)  // Temperature sensor: Parameter 5
        69 = 0 (Name=MOTOR_TEMPSENS_PAR6)  // Temperature sensor: Parameter 6
        70 = 0 (Name=MOTOR_TEMPSENS_PAR7)  // Temperature sensor: Parameter 7
        71 = 0 (Name=MOTOR_TEMPSENS_PAR8)  // Temperature sensor: Parameter 8
        72 = 0 (Name=MOTOR_TEMPSENS_PAR9)  // Temperature sensor: Parameter 9
        73 = 0 (Name=MOTOR_TEMPSENS_PAR10)  // Temperature sensor: Parameter 10
      Group  // Result Parameters of Parameter Identification
        47 = 1 (Name=MOTOR_POLEPAIRS)  // Motor: Number of pole-pairs
        48 = 0 (Name=MOTOR_VOLTAGE_RATED, Unit=V)  // Motor: Rated voltage
        49 = 1e-003 (Name=MOTOR_VOLTAGE_CONST, Unit=mV*min)  // Motor: Voltage constant
        50 = 500 (Name=MOTOR_SPEED_RATED, Unit=1/min)  // Motor: Rated speed
        51 = 500 (Name=MOTOR_SPEED_MAX, Unit=1/min)  // Motor: Maximum speed
        52 = 1e-003 (Name=MOTOR_TORQ_STALL, Unit=Nm)  // Motor: Stall torque
        53 = 1e-003 (Name=MOTOR_TORQ_RATED, Unit=Nm)  // Motor: Rated torque
        54 = 2e-003 (Name=MOTOR_TORQ_MAX, Unit=Nm)  // Motor: Peak torque
        55 = 1e-003 (Name=MOTOR_TORQ_CONST, Unit=Nm/A)  // Motor: Torque constant
        56 = 1e-003 (Name=MOTOR_CURR_STALL, Unit=A)  // Motor: Stall current
        57 = 1e-003 (Name=MOTOR_CURR_RATED, Unit=A)  // Motor: Rated current
        58 = 2e-003 (Name=MOTOR_CURR_MAX, Unit=A)  // Motor: Peak current
        59 = 0 (Name=MOTOR_WIND_CROSS_SECT, Unit=mm²)  // Motor: Line cross section
        60 = 1 (Name=MOTOR_STATOR_RESISTANCE, Unit=Ohm)  // Motor: Stator resistance
        61 = 1e-004 (Name=MOTOR_STATOR_INDUCTANCE, Unit=Henry)  // Motor: Stator inductance
        63 = 0 (Name=MOTOR_COMMUT_OFFSET, Unit=rad)  // Motor: Commutation offset
      Isolation parameters:
        74 = 0 (Name=MOTOR_WIND_TEMP_MAX, Unit=°C)  // Motor: Limit temperature
```

### Package Logical/30_MC/Libraries - Global libraries

### Library Logical/30_MC/Libraries/MotionLib (IEC, version 1.00.0)
Depends on: FiltLib, MpAxis, MpAlarmX, MpCom
